LIN {X 0,Y 418.23,Z 297.388,A -85,B 0,C 180,E1 -10312.167,E2 -10312.167} C_VEL
LIN {X 0,Y 418.144,Z 297.404,A -85,B 0,C 180,E1 -10315.148,E2 -10315.148} C_VEL
LIN {X 0,Y 418.014,Z 297.572,A -85,B 0,C 180,E1 -10316.685,E2 -10316.685} C_VEL
LIN {X 0,Y 417.751,Z 304.24,A -85,B 0,C 180,E1 -10320.799,E2 -10320.799} C_VEL
LIN {X 0,Y 417.681,Z 309.464,A -85,B 0,C 180,E1 -10324.057,E2 -10324.057} C_VEL
LIN {X 0,Y 417.666,Z 315.525,A -85,B 0,C 180,E1 -10327.741,E2 -10327.741} C_VEL
LIN {X 0,Y 417.566,Z 321.841,A -85,B 0,C 180,E1 -10331.35,E2 -10331.35} C_VEL
LIN {X 0,Y 417.611,Z 324.668,A -85,B 0,C 180,E1 -10332.823,E2 -10332.823} C_VEL
LIN {X 0,Y 420.936,Z 337.978,A -85,B 0,C 180,E1 -10333.371,E2 -10333.371} C_VEL
LIN {X 0,Y 422.449,Z 346.002,A -85,B 0,C 180,E1 -10333.786,E2 -10333.786} C_VEL
LIN {X 0,Y 421.995,Z 357.531,A -85,B 0,C 180,E1 -10334.426,E2 -10334.426} C_VEL
LIN {X 0,Y 421.355,Z 369.434,A -85,B 0,C 180,E1 -10335.289,E2 -10335.289} C_VEL
LIN {X 0,Y 420.762,Z 379.905,A -85,B 0,C 180,E1 -10336.264,E2 -10336.264} C_VEL
LIN {X 0,Y 419.975,Z 390.066,A -85,B 0,C 180,E1 -10337.435,E2 -10337.435} C_VEL
LIN {X 0,Y 419.339,Z 398.59,A -85,B 0,C 180,E1 -10338.643,E2 -10338.643} C_VEL
LIN {X 0,Y 418.753,Z 406.88,A -85,B 0,C 180,E1 -10340.094,E2 -10340.094} C_VEL
LIN {X 0,Y 418.261,Z 412.53,A -85,B 0,C 180,E1 -10341.302,E2 -10341.302} C_VEL
LIN {X 0,Y 417.846,Z 418.534,A -85,B 0,C 180,E1 -10342.913,E2 -10342.913} C_VEL
LIN {X 0,Y 417.439,Z 423.536,A -85,B 0,C 180,E1 -10344.687,E2 -10344.687} C_VEL
LIN {X 0,Y 417.442,Z 426.435,A -85,B 0,C 180,E1 -10346.139,E2 -10346.139} C_VEL
LIN {X 0,Y 417.313,Z 427.849,A -85,B 0,C 180,E1 -10347.104,E2 -10347.104} C_VEL
LIN {X 0,Y 417.143,Z 429.456,A -85,B 0,C 180,E1 -10349.035,E2 -10349.035} C_VEL
LIN {X 0,Y 417.142,Z 429.69,A -85,B 0,C 180,E1 -10350,E2 -10350} C_VEL
LIN {X 0,Y 417.135,Z 429.529,A -85,B 0,C 180,E1 -10350.822,E2 -10350.822} C_VEL
LIN {X 0,Y 416.515,Z 429.25,A -85,B 0,C 180,E1 -10351.629,E2 -10351.629} C_VEL
LIN {X 0,Y 413.745,Z 428.239,A -85,B 0,C 180,E1 -10352.936,E2 -10352.936} C_VEL
LIN {X 0,Y 411.4,Z 426.873,A -85,B 0,C 180,E1 -10353.98,E2 -10353.98} C_VEL
LIN {X 0,Y 410.41,Z 425.491,A -85,B 0,C 180,E1 -10354.775,E2 -10354.775} C_VEL
LIN {X 0,Y 410.339,Z 424.938,A -85,B 0,C 180,E1 -10355.041,E2 -10355.041} C_VEL
LIN {X 0,Y 410.76,Z 420.293,A -85,B 0,C 180,E1 -10356.879,E2 -10356.879} C_VEL
LIN {X 0,Y 411.059,Z 415.281,A -85,B 0,C 180,E1 -10358.356,E2 -10358.356} C_VEL
LIN {X 0,Y 411.623,Z 408.945,A -85,B 0,C 180,E1 -10359.831,E2 -10359.831} C_VEL
LIN {X 0,Y 412.235,Z 401.072,A -85,B 0,C 180,E1 -10361.307,E2 -10361.307} C_VEL
LIN {X 0,Y 412.91,Z 393.024,A -85,B 0,C 180,E1 -10362.534,E2 -10362.534} C_VEL
LIN {X 0,Y 413.699,Z 383.148,A -85,B 0,C 180,E1 -10363.759,E2 -10363.759} C_VEL
LIN {X 0,Y 414.35,Z 372.025,A -85,B 0,C 180,E1 -10364.865,E2 -10364.865} C_VEL
LIN {X 0,Y 415.089,Z 361.127,A -85,B 0,C 180,E1 -10365.718,E2 -10365.718} C_VEL
LIN {X 0,Y 415.573,Z 349.447,A -85,B 0,C 180,E1 -10366.428,E2 -10366.428} C_VEL
LIN {X 0,Y 415.517,Z 345.816,A -85,B 0,C 180,E1 -10366.618,E2 -10366.618} C_VEL
LIN {X 0,Y 412.954,Z 334.164,A -85,B 0,C 180,E1 -10367.215,E2 -10367.215} C_VEL
LIN {X 0,Y 410.545,Z 324.943,A -85,B 0,C 180,E1 -10367.581,E2 -10367.581} C_VEL
LIN {X 0,Y 410.556,Z 320.487,A -85,B 0,C 180,E1 -10370.021,E2 -10370.021} C_VEL
LIN {X 0,Y 410.607,Z 315.08,A -85,B 0,C 180,E1 -10373.183,E2 -10373.183} C_VEL
LIN {X 0,Y 410.646,Z 309.763,A -85,B 0,C 180,E1 -10376.422,E2 -10376.422} C_VEL
LIN {X 0,Y 410.701,Z 304.45,A -85,B 0,C 180,E1 -10379.753,E2 -10379.753} C_VEL
LIN {X 0,Y 411.026,Z 298.292,A -85,B 0,C 180,E1 -10383.612,E2 -10383.612} C_VEL
LIN {X 0,Y 411.186,Z 298.268,A -85,B 0,C 180,E1 -10386.743,E2 -10386.743} C_VEL
LIN {X 0,Y 411.215,Z 298.265,A -85,B 0,C 180,E1 -10389.728,E2 -10389.728} C_VEL
LIN {X 0,Y 411.176,Z 298.27,A -85,B 0,C 180,E1 -10393.134,E2 -10393.134} C_VEL
LIN {X 0,Y 411.17,Z 298.27,A -85,B 0,C 180,E1 -10395.881,E2 -10395.881} C_VEL
LIN {X 0,Y 411.167,Z 298.268,A -85,B 0,C 180,E1 -10398.772,E2 -10398.772} C_VEL
LIN {X 0,Y 411.208,Z 298.262,A -85,B 0,C 180,E1 -10401.831,E2 -10401.831} C_VEL
LIN {X 0,Y 411.091,Z 298.276,A -85,B 0,C 180,E1 -10405.146,E2 -10405.146} C_VEL
LIN {X 0,Y 410.886,Z 298.336,A -85,B 0,C 180,E1 -10407.029,E2 -10407.029} C_VEL
LIN {X 0,Y 410.68,Z 304.557,A -85,B 0,C 180,E1 -10410.782,E2 -10410.782} C_VEL
LIN {X 0,Y 410.578,Z 309.184,A -85,B 0,C 180,E1 -10413.573,E2 -10413.573} C_VEL
LIN {X 0,Y 410.571,Z 312.781,A -85,B 0,C 180,E1 -10415.743,E2 -10415.743} C_VEL
LIN {X 0,Y 410.522,Z 318.015,A -85,B 0,C 180,E1 -10418.93,E2 -10418.93} C_VEL
LIN {X 0,Y 410.439,Z 323.255,A -85,B 0,C 180,E1 -10422.048,E2 -10422.048} C_VEL
LIN {X 0,Y 410.453,Z 325.126,A -85,B 0,C 180,E1 -10423.157,E2 -10423.157} C_VEL
LIN {X 0,Y 413.417,Z 339.31,A -85,B 0,C 180,E1 -10423.77,E2 -10423.77} C_VEL
LIN {X 0,Y 414.485,Z 345.44,A -85,B 0,C 180,E1 -10424.097,E2 -10424.097} C_VEL
LIN {X 0,Y 413.983,Z 356.751,A -85,B 0,C 180,E1 -10424.744,E2 -10424.744} C_VEL
LIN {X 0,Y 413.372,Z 368.988,A -85,B 0,C 180,E1 -10425.651,E2 -10425.651} C_VEL
LIN {X 0,Y 412.891,Z 380.326,A -85,B 0,C 180,E1 -10426.715,E2 -10426.715} C_VEL
LIN {X 0,Y 412.187,Z 390.845,A -85,B 0,C 180,E1 -10427.944,E2 -10427.944} C_VEL
LIN {X 0,Y 411.694,Z 399.473,A -85,B 0,C 180,E1 -10429.177,E2 -10429.177} C_VEL
LIN {X 0,Y 411.18,Z 407.897,A -85,B 0,C 180,E1 -10430.655,E2 -10430.655} C_VEL
LIN {X 0,Y 410.759,Z 414.655,A -85,B 0,C 180,E1 -10432.133,E2 -10432.133} C_VEL
LIN {X 0,Y 410.528,Z 420.608,A -85,B 0,C 180,E1 -10433.783,E2 -10433.783} C_VEL
LIN {X 0,Y 410.3,Z 424.235,A -85,B 0,C 180,E1 -10435.087,E2 -10435.087} C_VEL
LIN {X 0,Y 410.357,Z 426.377,A -85,B 0,C 180,E1 -10436.072,E2 -10436.072} C_VEL
LIN {X 0,Y 410.249,Z 428.088,A -85,B 0,C 180,E1 -10437.054,E2 -10437.054} C_VEL
LIN {X 0,Y 410.135,Z 429.383,A -85,B 0,C 180,E1 -10438.036,E2 -10438.036} C_VEL
LIN {X 0,Y 410.089,Z 430.201,A -85,B 0,C 180,E1 -10439.018,E2 -10439.018} C_VEL
LIN {X 0,Y 410.102,Z 430.614,A -85,B 0,C 180,E1 -10440,E2 -10440} C_VEL
LIN {X 0,Y 410.136,Z 430.622,A -85,B 0,C 180,E1 -10440.982,E2 -10440.982} C_VEL
LIN {X 0,Y 410.22,Z 430.164,A -85,B 0,C 180,E1 -10441.964,E2 -10441.964} C_VEL
LIN {X 0,Y 410.309,Z 429.298,A -85,B 0,C 180,E1 -10442.945,E2 -10442.945} C_VEL
LIN {X 0,Y 410.419,Z 428.027,A -85,B 0,C 180,E1 -10443.928,E2 -10443.928} C_VEL
LIN {X 0,Y 410.502,Z 425.256,A -85,B 0,C 180,E1 -10445.403,E2 -10445.403} C_VEL
LIN {X 0,Y 410.839,Z 421.383,A -85,B 0,C 180,E1 -10446.877,E2 -10446.877} C_VEL
LIN {X 0,Y 411.196,Z 416.313,A -85,B 0,C 180,E1 -10448.353,E2 -10448.353} C_VEL
LIN {X 0,Y 411.729,Z 409.882,A -85,B 0,C 180,E1 -10449.828,E2 -10449.828} C_VEL
LIN {X 0,Y 412.317,Z 401.876,A -85,B 0,C 180,E1 -10451.304,E2 -10451.304} C_VEL
LIN {X 0,Y 412.986,Z 391.822,A -85,B 0,C 180,E1 -10452.781,E2 -10452.781} C_VEL
LIN {X 0,Y 413.808,Z 382.015,A -85,B 0,C 180,E1 -10453.93,E2 -10453.93} C_VEL
LIN {X 0,Y 414.435,Z 371.233,A -85,B 0,C 180,E1 -10454.962,E2 -10454.962} C_VEL
LIN {X 0,Y 415.113,Z 359.685,A -85,B 0,C 180,E1 -10455.842,E2 -10455.842} C_VEL
LIN {X 0,Y 415.727,Z 346.23,A -85,B 0,C 180,E1 -10456.636,E2 -10456.636} C_VEL
LIN {X 0,Y 412.949,Z 334.877,A -85,B 0,C 180,E1 -10457.308,E2 -10457.308} C_VEL
LIN {X 0,Y 410.978,Z 328.466,A -85,B 0,C 180,E1 -10457.662,E2 -10457.662} C_VEL
LIN {X 0,Y 411.017,Z 322.663,A -85,B 0,C 180,E1 -10461.044,E2 -10461.044} C_VEL
LIN {X 0,Y 411.115,Z 317.021,A -85,B 0,C 180,E1 -10464.222,E2 -10464.222} C_VEL
LIN {X 0,Y 411.206,Z 309.985,A -85,B 0,C 180,E1 -10468.035,E2 -10468.035} C_VEL
LIN {X 0,Y 411.401,Z 303.588,A -85,B 0,C 180,E1 -10471.333,E2 -10471.333} C_VEL
LIN {X 0,Y 411.353,Z 299.92,A -85,B 0,C 180,E1 -10473.157,E2 -10473.157} C_VEL
LIN {X 0,Y 411.094,Z 298.282,A -85,B 0,C 180,E1 -10474.048,E2 -10474.048} C_VEL
LIN {X 0,Y 411.188,Z 298.268,A -85,B 0,C 180,E1 -10476.742,E2 -10476.742} C_VEL
LIN {X 0,Y 411.211,Z 298.264,A -85,B 0,C 180,E1 -10479.727,E2 -10479.727} C_VEL
LIN {X 0,Y 411.173,Z 298.271,A -85,B 0,C 180,E1 -10483.134,E2 -10483.134} C_VEL
LIN {X 0,Y 411.227,Z 298.412,A -85,B 0,C 180,E1 -10485.594,E2 -10485.594} C_VEL
LIN {X 0,Y 412.81,Z 306.462,A -85,B 0,C 180,E1 -10489.143,E2 -10489.143} C_VEL
LIN {X 0,Y 414.03,Z 312.933,A -85,B 0,C 180,E1 -10491.865,E2 -10491.865} C_VEL
LIN {X 0,Y 414.518,Z 317.262,A -85,B 0,C 180,E1 -10493.6,E2 -10493.6} C_VEL
LIN {X 0,Y 413.908,Z 324.461,A -85,B 0,C 180,E1 -10496.305,E2 -10496.305} C_VEL
LIN {X 0,Y 413.168,Z 334.07,A -85,B 0,C 180,E1 -10499.811,E2 -10499.811} C_VEL
LIN {X 0,Y 412.443,Z 343.508,A -85,B 0,C 180,E1 -10503.156,E2 -10503.156} C_VEL
LIN {X 0,Y 411.875,Z 352.746,A -85,B 0,C 180,E1 -10506.36,E2 -10506.36} C_VEL
LIN {X 0,Y 411.304,Z 363.53,A -85,B 0,C 180,E1 -10510.017,E2 -10510.017} C_VEL
LIN {X 0,Y 410.937,Z 370.534,A -85,B 0,C 180,E1 -10512.357,E2 -10512.357} C_VEL
LIN {X 0,Y 413.007,Z 384.417,A -85,B 0,C 180,E1 -10512.886,E2 -10512.886} C_VEL
LIN {X 0,Y 414.755,Z 397.429,A -85,B 0,C 180,E1 -10513.574,E2 -10513.574} C_VEL
LIN {X 0,Y 414.347,Z 408.316,A -85,B 0,C 180,E1 -10514.253,E2 -10514.253} C_VEL
LIN {X 0,Y 413.464,Z 420.652,A -85,B 0,C 180,E1 -10515.228,E2 -10515.228} C_VEL
LIN {X 0,Y 412.7,Z 431.639,A -85,B 0,C 180,E1 -10516.333,E2 -10516.333} C_VEL
LIN {X 0,Y 411.963,Z 442.383,A -85,B 0,C 180,E1 -10517.687,E2 -10517.687} C_VEL
LIN {X 0,Y 411.291,Z 450.345,A -85,B 0,C 180,E1 -10518.917,E2 -10518.917} C_VEL
LIN {X 0,Y 410.814,Z 458.183,A -85,B 0,C 180,E1 -10520.398,E2 -10520.398} C_VEL
LIN {X 0,Y 410.483,Z 463.52,A -85,B 0,C 180,E1 -10521.632,E2 -10521.632} C_VEL
LIN {X 0,Y 410.253,Z 468.725,A -85,B 0,C 180,E1 -10523.113,E2 -10523.113} C_VEL
LIN {X 0,Y 410.147,Z 472.759,A -85,B 0,C 180,E1 -10524.592,E2 -10524.592} C_VEL
LIN {X 0,Y 409.992,Z 475.719,A -85,B 0,C 180,E1 -10526.068,E2 -10526.068} C_VEL
LIN {X 0,Y 410.083,Z 477.145,A -85,B 0,C 180,E1 -10527.053,E2 -10527.053} C_VEL
LIN {X 0,Y 410.097,Z 478.729,A -85,B 0,C 180,E1 -10529.018,E2 -10529.018} C_VEL
LIN {X 0,Y 410.07,Z 478.915,A -85,B 0,C 180,E1 -10530,E2 -10530} C_VEL
LIN {X 0,Y 410.099,Z 478.658,A -85,B 0,C 180,E1 -10530.982,E2 -10530.982} C_VEL
LIN {X 0,Y 410.087,Z 476.91,A -85,B 0,C 180,E1 -10532.947,E2 -10532.947} C_VEL
LIN {X 0,Y 410.013,Z 475.412,A -85,B 0,C 180,E1 -10533.932,E2 -10533.932} C_VEL
LIN {X 0,Y 410.175,Z 472.315,A -85,B 0,C 180,E1 -10535.407,E2 -10535.407} C_VEL
LIN {X 0,Y 410.253,Z 468.131,A -85,B 0,C 180,E1 -10536.887,E2 -10536.887} C_VEL
LIN {X 0,Y 410.574,Z 461.734,A -85,B 0,C 180,E1 -10538.614,E2 -10538.614} C_VEL
LIN {X 0,Y 410.954,Z 454.778,A -85,B 0,C 180,E1 -10540.096,E2 -10540.096} C_VEL
LIN {X 0,Y 411.525,Z 446.209,A -85,B 0,C 180,E1 -10541.576,E2 -10541.576} C_VEL
LIN {X 0,Y 412.128,Z 437.452,A -85,B 0,C 180,E1 -10542.808,E2 -10542.808} C_VEL
LIN {X 0,Y 412.75,Z 427.734,A -85,B 0,C 180,E1 -10543.938,E2 -10543.938} C_VEL
LIN {X 0,Y 413.534,Z 416.299,A -85,B 0,C 180,E1 -10545.021,E2 -10545.021} C_VEL
LIN {X 0,Y 414.379,Z 405.059,A -85,B 0,C 180,E1 -10545.872,E2 -10545.872} C_VEL
LIN {X 0,Y 414.735,Z 398.212,A -85,B 0,C 180,E1 -10546.3,E2 -10546.3} C_VEL
LIN {X 0,Y 413.023,Z 384.848,A -85,B 0,C 180,E1 -10547.066,E2 -10547.066} C_VEL
LIN {X 0,Y 411.421,Z 371.369,A -85,B 0,C 180,E1 -10547.642,E2 -10547.642} C_VEL
LIN {X 0,Y 410.851,Z 367.765,A -85,B 0,C 180,E1 -10547.781,E2 -10547.781} C_VEL
LIN {X 0,Y 411.229,Z 357.761,A -85,B 0,C 180,E1 -10551.032,E2 -10551.032} C_VEL
LIN {X 0,Y 411.705,Z 348.288,A -85,B 0,C 180,E1 -10554.186,E2 -10554.186} C_VEL
LIN {X 0,Y 412.237,Z 338.537,A -85,B 0,C 180,E1 -10557.561,E2 -10557.561} C_VEL
LIN {X 0,Y 413.002,Z 328.602,A -85,B 0,C 180,E1 -10561.211,E2 -10561.211} C_VEL
LIN {X 0,Y 413.835,Z 319.926,A -85,B 0,C 180,E1 -10564.675,E2 -10564.675} C_VEL
LIN {X 0,Y 414.252,Z 315.928,A -85,B 0,C 180,E1 -10566.427,E2 -10566.427} C_VEL
LIN {X 0,Y 413.761,Z 311.596,A -85,B 0,C 180,E1 -10568.616,E2 -10568.616} C_VEL
LIN {X 0,Y 412.864,Z 306.663,A -85,B 0,C 180,E1 -10571.597,E2 -10571.597} C_VEL
LIN {X 0,Y 412.142,Z 303.106,A -85,B 0,C 180,E1 -10574.359,E2 -10574.359} C_VEL
LIN {X 0,Y 411.617,Z 300.463,A -85,B 0,C 180,E1 -10577.239,E2 -10577.239} C_VEL
LIN {X 0,Y 411.295,Z 298.828,A -85,B 0,C 180,E1 -10580.259,E2 -10580.259} C_VEL
LIN {X 0,Y 411.192,Z 298.267,A -85,B 0,C 180,E1 -10583.258,E2 -10583.258} C_VEL
LIN {X 0,Y 411.214,Z 298.311,A -85,B 0,C 180,E1 -10585.667,E2 -10585.667} C_VEL
LIN {X 0,Y 411.347,Z 299.206,A -85,B 0,C 180,E1 -10589.165,E2 -10589.165} C_VEL
LIN {X 0,Y 411.635,Z 300.67,A -85,B 0,C 180,E1 -10592.601,E2 -10592.601} C_VEL
LIN {X 0,Y 411.738,Z 302.464,A -85,B 0,C 180,E1 -10595.817,E2 -10595.817} C_VEL
LIN {X 0,Y 411.703,Z 303.825,A -85,B 0,C 180,E1 -10597.941,E2 -10597.941} C_VEL
LIN {X 0,Y 411.545,Z 306.033,A -85,B 0,C 180,E1 -10601.067,E2 -10601.067} C_VEL
LIN {X 0,Y 411.46,Z 307.135,A -85,B 0,C 180,E1 -10602.467,E2 -10602.467} C_VEL
LIN {X 0,Y 415.682,Z 319.179,A -85,B 0,C 180,E1 -10603.227,E2 -10603.227} C_VEL
LIN {X 0,Y 416.32,Z 321.604,A -85,B 0,C 180,E1 -10603.386,E2 -10603.386} C_VEL
LIN {X 0,Y 415.851,Z 333.205,A -85,B 0,C 180,E1 -10604.06,E2 -10604.06} C_VEL
LIN {X 0,Y 415.147,Z 345.588,A -85,B 0,C 180,E1 -10604.989,E2 -10604.989} C_VEL
LIN {X 0,Y 414.484,Z 356.455,A -85,B 0,C 180,E1 -10606.018,E2 -10606.018} C_VEL
LIN {X 0,Y 413.726,Z 366.834,A -85,B 0,C 180,E1 -10607.242,E2 -10607.242} C_VEL
LIN {X 0,Y 413.091,Z 375.295,A -85,B 0,C 180,E1 -10608.469,E2 -10608.469} C_VEL
LIN {X 0,Y 412.405,Z 383.502,A -85,B 0,C 180,E1 -10609.94,E2 -10609.94} C_VEL
LIN {X 0,Y 411.874,Z 390.158,A -85,B 0,C 180,E1 -10611.438,E2 -10611.438} C_VEL
LIN {X 0,Y 411.474,Z 394.915,A -85,B 0,C 180,E1 -10612.777,E2 -10612.777} C_VEL
LIN {X 0,Y 411.056,Z 398.678,A -85,B 0,C 180,E1 -10614.112,E2 -10614.112} C_VEL
LIN {X 0,Y 411.018,Z 400.837,A -85,B 0,C 180,E1 -10615.096,E2 -10615.096} C_VEL
LIN {X 0,Y 410.772,Z 402.572,A -85,B 0,C 180,E1 -10616.076,E2 -10616.076} C_VEL
LIN {X 0,Y 410.511,Z 403.832,A -85,B 0,C 180,E1 -10617.056,E2 -10617.056} C_VEL
LIN {X 0,Y 410.347,Z 404.677,A -85,B 0,C 180,E1 -10618.037,E2 -10618.037} C_VEL
LIN {X 0,Y 410.276,Z 405.113,A -85,B 0,C 180,E1 -10619.019,E2 -10619.019} C_VEL
LIN {X 0,Y 410.241,Z 405.1,A -85,B 0,C 180,E1 -10620,E2 -10620} C_VEL
LIN {X 0,Y 410.244,Z 404.668,A -85,B 0,C 180,E1 -10620.982,E2 -10620.982} C_VEL
LIN {X 0,Y 410.318,Z 403.834,A -85,B 0,C 180,E1 -10621.963,E2 -10621.963} C_VEL
LIN {X 0,Y 410.497,Z 402.572,A -85,B 0,C 180,E1 -10622.944,E2 -10622.944} C_VEL
LIN {X 0,Y 410.733,Z 399.85,A -85,B 0,C 180,E1 -10624.416,E2 -10624.416} C_VEL
LIN {X 0,Y 410.758,Z 396.102,A -85,B 0,C 180,E1 -10625.892,E2 -10625.892} C_VEL
LIN {X 0,Y 411.045,Z 391.08,A -85,B 0,C 180,E1 -10627.395,E2 -10627.395} C_VEL
LIN {X 0,Y 411.456,Z 383.804,A -85,B 0,C 180,E1 -10629.091,E2 -10629.091} C_VEL
LIN {X 0,Y 411.933,Z 375.802,A -85,B 0,C 180,E1 -10630.568,E2 -10630.568} C_VEL
LIN {X 0,Y 412.561,Z 365.797,A -85,B 0,C 180,E1 -10632.045,E2 -10632.045} C_VEL
LIN {X 0,Y 413.175,Z 355.451,A -85,B 0,C 180,E1 -10633.275,E2 -10633.275} C_VEL
LIN {X 0,Y 413.759,Z 343.258,A -85,B 0,C 180,E1 -10634.435,E2 -10634.435} C_VEL
LIN {X 0,Y 414.217,Z 332.568,A -85,B 0,C 180,E1 -10635.248,E2 -10635.248} C_VEL
LIN {X 0,Y 414.783,Z 319.92,A -85,B 0,C 180,E1 -10635.988,E2 -10635.988} C_VEL
LIN {X 0,Y 414.081,Z 315.24,A -85,B 0,C 180,E1 -10636.243,E2 -10636.243} C_VEL
LIN {X 0,Y 410.732,Z 301.39,A -85,B 0,C 180,E1 -10636.892,E2 -10636.892} C_VEL
LIN {X 0,Y 410.516,Z 300.22,A -85,B 0,C 180,E1 -10636.952,E2 -10636.952} C_VEL
LIN {X 0,Y 410.442,Z 299.006,A -85,B 0,C 180,E1 -10637.952,E2 -10637.952} C_VEL
LIN {X 0,Y 410.56,Z 298.347,A -85,B 0,C 180,E1 -10638.98,E2 -10638.98} C_VEL
LIN {X 0,Y 410.936,Z 298.298,A -85,B 0,C 180,E1 -10642.551,E2 -10642.551} C_VEL
LIN {X 0,Y 411.164,Z 298.264,A -85,B 0,C 180,E1 -10645.298,E2 -10645.298} C_VEL
LIN {X 0,Y 411.243,Z 298.254,A -85,B 0,C 180,E1 -10647.479,E2 -10647.479} C_VEL
LIN {X 0,Y 411.192,Z 298.26,A -85,B 0,C 180,E1 -10650.848,E2 -10650.848} C_VEL
LIN {X 0,Y 411.209,Z 298.263,A -85,B 0,C 180,E1 -10654.333,E2 -10654.333} C_VEL
LIN {X 0,Y 411.197,Z 298.269,A -85,B 0,C 180,E1 -10657.974,E2 -10657.974} C_VEL
LIN {X 0,Y 411.166,Z 298.269,A -85,B 0,C 180,E1 -10661.228,E2 -10661.228} C_VEL
LIN {X 0,Y 411.18,Z 298.265,A -85,B 0,C 180,E1 -10664.49,E2 -10664.49} C_VEL
LIN {X 0,Y 411.18,Z 298.266,A -85,B 0,C 180,E1 -10668.195,E2 -10668.195} C_VEL
LIN {X 0,Y 411.22,Z 298.261,A -85,B 0,C 180,E1 -10670.776,E2 -10670.776} C_VEL
LIN {X 0,Y 411.187,Z 298.269,A -85,B 0,C 180,E1 -10673.449,E2 -10673.449} C_VEL
LIN {X 0,Y 410.989,Z 298.381,A -85,B 0,C 180,E1 -10676.604,E2 -10676.604} C_VEL
LIN {X 0,Y 410.732,Z 305.091,A -85,B 0,C 180,E1 -10680.769,E2 -10680.769} C_VEL
LIN {X 0,Y 410.646,Z 309.599,A -85,B 0,C 180,E1 -10683.578,E2 -10683.578} C_VEL
LIN {X 0,Y 410.607,Z 314.889,A -85,B 0,C 180,E1 -10686.817,E2 -10686.817} C_VEL
LIN {X 0,Y 410.595,Z 320.851,A -85,B 0,C 180,E1 -10690.291,E2 -10690.291} C_VEL
LIN {X 0,Y 410.564,Z 324.92,A -85,B 0,C 180,E1 -10692.504,E2 -10692.504} C_VEL
LIN {X 0,Y 414.246,Z 339.604,A -85,B 0,C 180,E1 -10693.142,E2 -10693.142} C_VEL
LIN {X 0,Y 415.607,Z 347.386,A -85,B 0,C 180,E1 -10693.563,E2 -10693.563} C_VEL
LIN {X 0,Y 415.087,Z 359.759,A -85,B 0,C 180,E1 -10694.282,E2 -10694.282} C_VEL
LIN {X 0,Y 414.393,Z 371.394,A -85,B 0,C 180,E1 -10695.175,E2 -10695.175} C_VEL
LIN {X 0,Y 413.71,Z 382.276,A -85,B 0,C 180,E1 -10696.242,E2 -10696.242} C_VEL
LIN {X 0,Y 412.944,Z 392.35,A -85,B 0,C 180,E1 -10697.467,E2 -10697.467} C_VEL
LIN {X 0,Y 412.185,Z 401.962,A -85,B 0,C 180,E1 -10698.941,E2 -10698.941} C_VEL
LIN {X 0,Y 411.537,Z 409.688,A -85,B 0,C 180,E1 -10700.415,E2 -10700.415} C_VEL
LIN {X 0,Y 411.119,Z 414.904,A -85,B 0,C 180,E1 -10701.645,E2 -10701.645} C_VEL
LIN {X 0,Y 410.76,Z 420,A -85,B 0,C 180,E1 -10703.121,E2 -10703.121} C_VEL
LIN {X 0,Y 410.383,Z 423.951,A -85,B 0,C 180,E1 -10704.595,E2 -10704.595} C_VEL
LIN {X 0,Y 410.386,Z 426.85,A -85,B 0,C 180,E1 -10706.072,E2 -10706.072} C_VEL
LIN {X 0,Y 410.25,Z 428.264,A -85,B 0,C 180,E1 -10707.054,E2 -10707.054} C_VEL
LIN {X 0,Y 410.062,Z 429.871,A -85,B 0,C 180,E1 -10709.018,E2 -10709.018} C_VEL
LIN {X 0,Y 410.057,Z 430.104,A -85,B 0,C 180,E1 -10710,E2 -10710} C_VEL
LIN {X 0,Y 410.135,Z 429.332,A -85,B 0,C 180,E1 -10711.964,E2 -10711.964} C_VEL
LIN {X 0,Y 410.249,Z 428.368,A -85,B 0,C 180,E1 -10712.946,E2 -10712.946} C_VEL
LIN {X 0,Y 410.378,Z 427.012,A -85,B 0,C 180,E1 -10713.928,E2 -10713.928} C_VEL
LIN {X 0,Y 410.339,Z 424.938,A -85,B 0,C 180,E1 -10715.041,E2 -10715.041} C_VEL
LIN {X 0,Y 409.757,Z 423.224,A -85,B 0,C 180,E1 -10715.828,E2 -10715.828} C_VEL
LIN {X 0,Y 407.185,Z 420.047,A -85,B 0,C 180,E1 -10717.097,E2 -10717.097} C_VEL
LIN {X 0,Y 404.697,Z 416.203,A -85,B 0,C 180,E1 -10718.34,E2 -10718.34} C_VEL
LIN {X 0,Y 404.251,Z 413.42,A -85,B 0,C 180,E1 -10719.078,E2 -10719.078} C_VEL
LIN {X 0,Y 404.867,Z 406.94,A -85,B 0,C 180,E1 -10720.502,E2 -10720.502} C_VEL
LIN {X 0,Y 405.569,Z 398.435,A -85,B 0,C 180,E1 -10722.002,E2 -10722.002} C_VEL
LIN {X 0,Y 406.367,Z 389.716,A -85,B 0,C 180,E1 -10723.247,E2 -10723.247} C_VEL
LIN {X 0,Y 407.019,Z 380.308,A -85,B 0,C 180,E1 -10724.354,E2 -10724.354} C_VEL
LIN {X 0,Y 407.695,Z 369.564,A -85,B 0,C 180,E1 -10725.369,E2 -10725.369} C_VEL
LIN {X 0,Y 408.447,Z 358.139,A -85,B 0,C 180,E1 -10726.213,E2 -10726.213} C_VEL
LIN {X 0,Y 408.727,Z 347.121,A -85,B 0,C 180,E1 -10726.853,E2 -10726.853} C_VEL
LIN {X 0,Y 405.966,Z 334.5,A -85,B 0,C 180,E1 -10727.521,E2 -10727.521} C_VEL
LIN {X 0,Y 403.51,Z 325.248,A -85,B 0,C 180,E1 -10727.928,E2 -10727.928} C_VEL
LIN {X 0,Y 403.501,Z 320.783,A -85,B 0,C 180,E1 -10730.387,E2 -10730.387} C_VEL
LIN {X 0,Y 403.562,Z 315.298,A -85,B 0,C 180,E1 -10733.612,E2 -10733.612} C_VEL
LIN {X 0,Y 403.638,Z 309.177,A -85,B 0,C 180,E1 -10737.377,E2 -10737.377} C_VEL
LIN {X 0,Y 403.7,Z 304.485,A -85,B 0,C 180,E1 -10740.322,E2 -10740.322} C_VEL
LIN {X 0,Y 403.995,Z 299.167,A -85,B 0,C 180,E1 -10743.688,E2 -10743.688} C_VEL
LIN {X 0,Y 404.133,Z 299.147,A -85,B 0,C 180,E1 -10746.874,E2 -10746.874} C_VEL
LIN {X 0,Y 404.15,Z 299.145,A -85,B 0,C 180,E1 -10750.08,E2 -10750.08} C_VEL
LIN {X 0,Y 404.155,Z 299.145,A -85,B 0,C 180,E1 -10753.084,E2 -10753.084} C_VEL
LIN {X 0,Y 404.15,Z 299.144,A -85,B 0,C 180,E1 -10755.926,E2 -10755.926} C_VEL
LIN {X 0,Y 404.122,Z 299.146,A -85,B 0,C 180,E1 -10758.635,E2 -10758.635} C_VEL
LIN {X 0,Y 404.157,Z 299.14,A -85,B 0,C 180,E1 -10761.492,E2 -10761.492} C_VEL
LIN {X 0,Y 404.058,Z 299.152,A -85,B 0,C 180,E1 -10764.971,E2 -10764.971} C_VEL
LIN {X 0,Y 403.845,Z 299.325,A -85,B 0,C 180,E1 -10767.109,E2 -10767.109} C_VEL
LIN {X 0,Y 403.628,Z 305.437,A -85,B 0,C 180,E1 -10770.821,E2 -10770.821} C_VEL
LIN {X 0,Y 403.514,Z 310.989,A -85,B 0,C 180,E1 -10774.187,E2 -10774.187} C_VEL
LIN {X 0,Y 403.484,Z 316.391,A -85,B 0,C 180,E1 -10777.468,E2 -10777.468} C_VEL
LIN {X 0,Y 403.459,Z 321.702,A -85,B 0,C 180,E1 -10780.672,E2 -10780.672} C_VEL
LIN {X 0,Y 403.396,Z 325.469,A -85,B 0,C 180,E1 -10782.931,E2 -10782.931} C_VEL
LIN {X 0,Y 405.999,Z 337.78,A -85,B 0,C 180,E1 -10783.455,E2 -10783.455} C_VEL
LIN {X 0,Y 407.556,Z 346.315,A -85,B 0,C 180,E1 -10783.918,E2 -10783.918} C_VEL
LIN {X 0,Y 407.015,Z 357.948,A -85,B 0,C 180,E1 -10784.604,E2 -10784.604} C_VEL
LIN {X 0,Y 406.312,Z 370.998,A -85,B 0,C 180,E1 -10785.613,E2 -10785.613} C_VEL
LIN {X 0,Y 405.788,Z 382.335,A -85,B 0,C 180,E1 -10786.733,E2 -10786.733} C_VEL
LIN {X 0,Y 405.08,Z 392.598,A -85,B 0,C 180,E1 -10787.983,E2 -10787.983} C_VEL
LIN {X 0,Y 404.595,Z 401.012,A -85,B 0,C 180,E1 -10789.238,E2 -10789.238} C_VEL
LIN {X 0,Y 404.076,Z 409.206,A -85,B 0,C 180,E1 -10790.742,E2 -10790.742} C_VEL
LIN {X 0,Y 403.735,Z 414.81,A -85,B 0,C 180,E1 -10791.995,E2 -10791.995} C_VEL
LIN {X 0,Y 403.494,Z 420.111,A -85,B 0,C 180,E1 -10793.45,E2 -10793.45} C_VEL
LIN {X 0,Y 403.231,Z 424.518,A -85,B 0,C 180,E1 -10795,E2 -10795} C_VEL
LIN {X 0,Y 403.272,Z 426.71,A -85,B 0,C 180,E1 -10796.003,E2 -10796.003} C_VEL
LIN {X 0,Y 403.188,Z 428.443,A -85,B 0,C 180,E1 -10797.002,E2 -10797.002} C_VEL
LIN {X 0,Y 403.064,Z 429.768,A -85,B 0,C 180,E1 -10798.001,E2 -10798.001} C_VEL
LIN {X 0,Y 403.009,Z 430.626,A -85,B 0,C 180,E1 -10799.001,E2 -10799.001} C_VEL
LIN {X 0,Y 403.018,Z 431.061,A -85,B 0,C 180,E1 -10800,E2 -10800} C_VEL
LIN {X 0,Y 403.053,Z 431.099,A -85,B 0,C 180,E1 -10800.999,E2 -10800.999} C_VEL
LIN {X 0,Y 403.143,Z 430.678,A -85,B 0,C 180,E1 -10801.998,E2 -10801.998} C_VEL
LIN {X 0,Y 403.245,Z 429.832,A -85,B 0,C 180,E1 -10802.997,E2 -10802.997} C_VEL
LIN {X 0,Y 403.373,Z 428.581,A -85,B 0,C 180,E1 -10803.996,E2 -10803.996} C_VEL
LIN {X 0,Y 403.456,Z 425.848,A -85,B 0,C 180,E1 -10805.498,E2 -10805.498} C_VEL
LIN {X 0,Y 403.892,Z 421.002,A -85,B 0,C 180,E1 -10807.323,E2 -10807.323} C_VEL
LIN {X 0,Y 404.409,Z 415.048,A -85,B 0,C 180,E1 -10808.998,E2 -10808.998} C_VEL
LIN {X 0,Y 404.977,Z 408.173,A -85,B 0,C 180,E1 -10810.499,E2 -10810.499} C_VEL
LIN {X 0,Y 405.638,Z 399.612,A -85,B 0,C 180,E1 -10812,E2 -10812} C_VEL
LIN {X 0,Y 406.383,Z 390.763,A -85,B 0,C 180,E1 -10813.247,E2 -10813.247} C_VEL
LIN {X 0,Y 407.212,Z 379.809,A -85,B 0,C 180,E1 -10814.507,E2 -10814.507} C_VEL
LIN {X 0,Y 407.88,Z 369.209,A -85,B 0,C 180,E1 -10815.49,E2 -10815.49} C_VEL
LIN {X 0,Y 408.594,Z 357.572,A -85,B 0,C 180,E1 -10816.348,E2 -10816.348} C_VEL
LIN {X 0,Y 409.123,Z 348.106,A -85,B 0,C 180,E1 -10816.902,E2 -10816.902} C_VEL
LIN {X 0,Y 406.438,Z 336.838,A -85,B 0,C 180,E1 -10817.611,E2 -10817.611} C_VEL
LIN {X 0,Y 403.997,Z 329.018,A -85,B 0,C 180,E1 -10818.084,E2 -10818.084} C_VEL
LIN {X 0,Y 404.04,Z 325.149,A -85,B 0,C 180,E1 -10820.358,E2 -10820.358} C_VEL
LIN {X 0,Y 404.125,Z 319.566,A -85,B 0,C 180,E1 -10823.577,E2 -10823.577} C_VEL
LIN {X 0,Y 404.197,Z 313.631,A -85,B 0,C 180,E1 -10826.877,E2 -10826.877} C_VEL
LIN {X 0,Y 404.426,Z 307.299,A -85,B 0,C 180,E1 -10830.262,E2 -10830.262} C_VEL
LIN {X 0,Y 404.524,Z 302.761,A -85,B 0,C 180,E1 -10832.587,E2 -10832.587} C_VEL
LIN {X 0,Y 404.066,Z 299.158,A -85,B 0,C 180,E1 -10834.573,E2 -10834.573} C_VEL
LIN {X 0,Y 404.142,Z 299.145,A -85,B 0,C 180,E1 -10837.492,E2 -10837.492} C_VEL
LIN {X 0,Y 404.149,Z 299.145,A -85,B 0,C 180,E1 -10840.08,E2 -10840.08} C_VEL
LIN {X 0,Y 404.152,Z 299.145,A -85,B 0,C 180,E1 -10843.083,E2 -10843.083} C_VEL
LIN {X 0,Y 404.169,Z 299.242,A -85,B 0,C 180,E1 -10845.213,E2 -10845.213} C_VEL
LIN {X 0,Y 405.442,Z 305.847,A -85,B 0,C 180,E1 -10848.191,E2 -10848.191} C_VEL
LIN {X 0,Y 406.979,Z 313.657,A -85,B 0,C 180,E1 -10851.561,E2 -10851.561} C_VEL
LIN {X 0,Y 407.556,Z 318.378,A -85,B 0,C 180,E1 -10853.492,E2 -10853.492} C_VEL
LIN {X 0,Y 406.848,Z 326.113,A -85,B 0,C 180,E1 -10856.442,E2 -10856.442} C_VEL
LIN {X 0,Y 406.11,Z 335.475,A -85,B 0,C 180,E1 -10859.915,E2 -10859.915} C_VEL
LIN {X 0,Y 405.265,Z 346.155,A -85,B 0,C 180,E1 -10863.755,E2 -10863.755} C_VEL
LIN {X 0,Y 404.805,Z 353.857,A -85,B 0,C 180,E1 -10866.465,E2 -10866.465} C_VEL
LIN {X 0,Y 404.165,Z 364.865,A -85,B 0,C 180,E1 -10870.275,E2 -10870.275} C_VEL
LIN {X 0,Y 403.901,Z 370.036,A -85,B 0,C 180,E1 -10872.043,E2 -10872.043} C_VEL
LIN {X 0,Y 406.085,Z 384.87,A -85,B 0,C 180,E1 -10872.63,E2 -10872.63} C_VEL
LIN {X 0,Y 407.787,Z 397.869,A -85,B 0,C 180,E1 -10873.35,E2 -10873.35} C_VEL
LIN {X 0,Y 407.74,Z 404.003,A -85,B 0,C 180,E1 -10873.734,E2 -10873.734} C_VEL
LIN {X 0,Y 406.885,Z 415.744,A -85,B 0,C 180,E1 -10874.599,E2 -10874.599} C_VEL
LIN {X 0,Y 406.074,Z 426.413,A -85,B 0,C 180,E1 -10875.594,E2 -10875.594} C_VEL
LIN {X 0,Y 405.387,Z 436.187,A -85,B 0,C 180,E1 -10876.722,E2 -10876.722} C_VEL
LIN {X 0,Y 404.672,Z 445.102,A -85,B 0,C 180,E1 -10877.971,E2 -10877.971} C_VEL
LIN {X 0,Y 403.999,Z 453.863,A -85,B 0,C 180,E1 -10879.475,E2 -10879.475} C_VEL
LIN {X 0,Y 403.56,Z 460.884,A -85,B 0,C 180,E1 -10880.983,E2 -10880.983} C_VEL
LIN {X 0,Y 403.211,Z 466.502,A -85,B 0,C 180,E1 -10882.488,E2 -10882.488} C_VEL
LIN {X 0,Y 403.069,Z 470.919,A -85,B 0,C 180,E1 -10883.995,E2 -10883.995} C_VEL
LIN {X 0,Y 403.044,Z 473.249,A -85,B 0,C 180,E1 -10884.998,E2 -10884.998} C_VEL
LIN {X 0,Y 402.912,Z 475.129,A -85,B 0,C 180,E1 -10885.999,E2 -10885.999} C_VEL
LIN {X 0,Y 403.018,Z 476.558,A -85,B 0,C 180,E1 -10887.001,E2 -10887.001} C_VEL
LIN {X 0,Y 403.044,Z 478.14,A -85,B 0,C 180,E1 -10889.001,E2 -10889.001} C_VEL
LIN {X 0,Y 403.018,Z 478.323,A -85,B 0,C 180,E1 -10890,E2 -10890} C_VEL
LIN {X 0,Y 403.047,Z 478.062,A -85,B 0,C 180,E1 -10890.999,E2 -10890.999} C_VEL
LIN {X 0,Y 403.024,Z 476.3,A -85,B 0,C 180,E1 -10892.999,E2 -10892.999} C_VEL
LIN {X 0,Y 402.933,Z 474.79,A -85,B 0,C 180,E1 -10894.001,E2 -10894.001} C_VEL
LIN {X 0,Y 403.093,Z 471.678,A -85,B 0,C 180,E1 -10895.503,E2 -10895.503} C_VEL
LIN {X 0,Y 403.186,Z 467.48,A -85,B 0,C 180,E1 -10897.009,E2 -10897.009} C_VEL
LIN {X 0,Y 403.527,Z 461.077,A -85,B 0,C 180,E1 -10898.766,E2 -10898.766} C_VEL
LIN {X 0,Y 403.896,Z 454.142,A -85,B 0,C 180,E1 -10900.274,E2 -10900.274} C_VEL
LIN {X 0,Y 404.508,Z 445.548,A -85,B 0,C 180,E1 -10901.78,E2 -10901.78} C_VEL
LIN {X 0,Y 405.181,Z 436.824,A -85,B 0,C 180,E1 -10903.032,E2 -10903.032} C_VEL
LIN {X 0,Y 405.868,Z 426.416,A -85,B 0,C 180,E1 -10904.26,E2 -10904.26} C_VEL
LIN {X 0,Y 406.755,Z 414.379,A -85,B 0,C 180,E1 -10905.406,E2 -10905.406} C_VEL
LIN {X 0,Y 407.631,Z 402.823,A -85,B 0,C 180,E1 -10906.27,E2 -10906.27} C_VEL
LIN {X 0,Y 407.735,Z 397.959,A -85,B 0,C 180,E1 -10906.588,E2 -10906.588} C_VEL
LIN {X 0,Y 406.238,Z 385.682,A -85,B 0,C 180,E1 -10907.328,E2 -10907.328} C_VEL
LIN {X 0,Y 404.678,Z 372.195,A -85,B 0,C 180,E1 -10907.951,E2 -10907.951} C_VEL
LIN {X 0,Y 403.813,Z 366.974,A -85,B 0,C 180,E1 -10908.162,E2 -10908.162} C_VEL
LIN {X 0,Y 404.22,Z 357.201,A -85,B 0,C 180,E1 -10911.415,E2 -10911.415} C_VEL
LIN {X 0,Y 404.724,Z 347.808,A -85,B 0,C 180,E1 -10914.63,E2 -10914.63} C_VEL
LIN {X 0,Y 405.268,Z 338.595,A -85,B 0,C 180,E1 -10917.919,E2 -10917.919} C_VEL
LIN {X 0,Y 406.025,Z 329.682,A -85,B 0,C 180,E1 -10921.284,E2 -10921.284} C_VEL
LIN {X 0,Y 407.053,Z 320.071,A -85,B 0,C 180,E1 -10925.265,E2 -10925.265} C_VEL
LIN {X 0,Y 407.292,Z 316.024,A -85,B 0,C 180,E1 -10927.153,E2 -10927.153} C_VEL
LIN {X 0,Y 406.504,Z 311.311,A -85,B 0,C 180,E1 -10929.769,E2 -10929.769} C_VEL
LIN {X 0,Y 405.725,Z 307.251,A -85,B 0,C 180,E1 -10932.498,E2 -10932.498} C_VEL
LIN {X 0,Y 405.105,Z 303.982,A -85,B 0,C 180,E1 -10935.34,E2 -10935.34} C_VEL
LIN {X 0,Y 404.636,Z 301.661,A -85,B 0,C 180,E1 -10938.319,E2 -10938.319} C_VEL
LIN {X 0,Y 404.393,Z 300.316,A -85,B 0,C 180,E1 -10941.45,E2 -10941.45} C_VEL
LIN {X 0,Y 404.324,Z 299.963,A -85,B 0,C 180,E1 -10944.782,E2 -10944.782} C_VEL
LIN {X 0,Y 404.412,Z 300.571,A -85,B 0,C 180,E1 -10948.38,E2 -10948.38} C_VEL
LIN {X 0,Y 404.565,Z 301.43,A -85,B 0,C 180,E1 -10950.895,E2 -10950.895} C_VEL
LIN {X 0,Y 404.734,Z 302.44,A -85,B 0,C 180,E1 -10953.161,E2 -10953.161} C_VEL
LIN {X 0,Y 404.763,Z 303.633,A -85,B 0,C 180,E1 -10955.372,E2 -10955.372} C_VEL
LIN {X 0,Y 404.742,Z 304.939,A -85,B 0,C 180,E1 -10957.542,E2 -10957.542} C_VEL
LIN {X 0,Y 404.587,Z 307.096,A -85,B 0,C 180,E1 -10960.728,E2 -10960.728} C_VEL
LIN {X 0,Y 404.53,Z 308.26,A -85,B 0,C 180,E1 -10962.064,E2 -10962.064} C_VEL
LIN {X 0,Y 409.001,Z 320.719,A -85,B 0,C 180,E1 -10962.909,E2 -10962.909} C_VEL
LIN {X 0,Y 409.718,Z 323.707,A -85,B 0,C 180,E1 -10963.11,E2 -10963.11} C_VEL
LIN {X 0,Y 409.085,Z 336.772,A -85,B 0,C 180,E1 -10963.917,E2 -10963.917} C_VEL
LIN {X 0,Y 408.329,Z 348.819,A -85,B 0,C 180,E1 -10964.885,E2 -10964.885} C_VEL
LIN {X 0,Y 407.511,Z 360.029,A -85,B 0,C 180,E1 -10966.028,E2 -10966.028} C_VEL
LIN {X 0,Y 406.746,Z 369.839,A -85,B 0,C 180,E1 -10967.273,E2 -10967.273} C_VEL
LIN {X 0,Y 406.089,Z 377.887,A -85,B 0,C 180,E1 -10968.52,E2 -10968.52} C_VEL
LIN {X 0,Y 405.323,Z 385.761,A -85,B 0,C 180,E1 -10970.015,E2 -10970.015} C_VEL
LIN {X 0,Y 404.861,Z 392.202,A -85,B 0,C 180,E1 -10971.565,E2 -10971.565} C_VEL
LIN {X 0,Y 404.255,Z 396.955,A -85,B 0,C 180,E1 -10973.01,E2 -10973.01} C_VEL
LIN {X 0,Y 404.035,Z 400.688,A -85,B 0,C 180,E1 -10974.51,E2 -10974.51} C_VEL
LIN {X 0,Y 403.746,Z 403.388,A -85,B 0,C 180,E1 -10976.007,E2 -10976.007} C_VEL
LIN {X 0,Y 403.473,Z 404.625,A -85,B 0,C 180,E1 -10977.005,E2 -10977.005} C_VEL
LIN {X 0,Y 403.296,Z 405.446,A -85,B 0,C 180,E1 -10978.003,E2 -10978.003} C_VEL
LIN {X 0,Y 403.217,Z 405.852,A -85,B 0,C 180,E1 -10979.001,E2 -10979.001} C_VEL
LIN {X 0,Y 403.18,Z 405.8,A -85,B 0,C 180,E1 -10980,E2 -10980} C_VEL
LIN {X 0,Y 403.186,Z 405.341,A -85,B 0,C 180,E1 -10980.999,E2 -10980.999} C_VEL
LIN {X 0,Y 403.269,Z 404.473,A -85,B 0,C 180,E1 -10981.998,E2 -10981.998} C_VEL
LIN {X 0,Y 403.457,Z 403.161,A -85,B 0,C 180,E1 -10982.996,E2 -10982.996} C_VEL
LIN {X 0,Y 403.673,Z 400.385,A -85,B 0,C 180,E1 -10984.494,E2 -10984.494} C_VEL
LIN {X 0,Y 403.701,Z 396.575,A -85,B 0,C 180,E1 -10985.996,E2 -10985.996} C_VEL
LIN {X 0,Y 404.047,Z 390.747,A -85,B 0,C 180,E1 -10987.718,E2 -10987.718} C_VEL
LIN {X 0,Y 404.455,Z 384.134,A -85,B 0,C 180,E1 -10989.249,E2 -10989.249} C_VEL
LIN {X 0,Y 404.941,Z 376.014,A -85,B 0,C 180,E1 -10990.753,E2 -10990.753} C_VEL
LIN {X 0,Y 405.592,Z 365.906,A -85,B 0,C 180,E1 -10992.255,E2 -10992.255} C_VEL
LIN {X 0,Y 406.244,Z 355.393,A -85,B 0,C 180,E1 -10993.506,E2 -10993.506} C_VEL
LIN {X 0,Y 406.789,Z 344.265,A -85,B 0,C 180,E1 -10994.58,E2 -10994.58} C_VEL
LIN {X 0,Y 407.326,Z 332.108,A -85,B 0,C 180,E1 -10995.512,E2 -10995.512} C_VEL
LIN {X 0,Y 407.847,Z 319.978,A -85,B 0,C 180,E1 -10996.225,E2 -10996.225} C_VEL
LIN {X 0,Y 404.876,Z 306.729,A -85,B 0,C 180,E1 -10996.923,E2 -10996.923} C_VEL
LIN {X 0,Y 403.486,Z 300.794,A -85,B 0,C 180,E1 -10997.181,E2 -10997.181} C_VEL
LIN {X 0,Y 403.408,Z 299.441,A -85,B 0,C 180,E1 -10998.276,E2 -10998.276} C_VEL
LIN {X 0,Y 403.658,Z 299.204,A -85,B 0,C 180,E1 -11000.378,E2 -11000.378} C_VEL
LIN {X 0,Y 403.98,Z 299.166,A -85,B 0,C 180,E1 -11003.586,E2 -11003.586} C_VEL
LIN {X 0,Y 404.137,Z 299.138,A -85,B 0,C 180,E1 -11005.77,E2 -11005.77} C_VEL
LIN {X 0,Y 404.189,Z 299.134,A -85,B 0,C 180,E1 -11008,E2 -11008} C_VEL
LIN {X 0,Y 404.142,Z 299.136,A -85,B 0,C 180,E1 -11011.558,E2 -11011.558} C_VEL
LIN {X 0,Y 404.187,Z 299.131,A -85,B 0,C 180,E1 -11015.016,E2 -11015.016} C_VEL
LIN {X 0,Y 404.157,Z 299.14,A -85,B 0,C 180,E1 -11018.757,E2 -11018.757} C_VEL
LIN {X 0,Y 404.126,Z 299.148,A -85,B 0,C 180,E1 -11021.6,E2 -11021.6} C_VEL
LIN {X 0,Y 404.15,Z 299.141,A -85,B 0,C 180,E1 -11024.522,E2 -11024.522} C_VEL
LIN {X 0,Y 404.139,Z 299.142,A -85,B 0,C 180,E1 -11027.296,E2 -11027.296} C_VEL
LIN {X 0,Y 404.171,Z 299.141,A -85,B 0,C 180,E1 -11029.955,E2 -11029.955} C_VEL
LIN {X 0,Y 404.133,Z 299.145,A -85,B 0,C 180,E1 -11033.126,E2 -11033.126} C_VEL
LIN {X 0,Y 403.973,Z 299.168,A -85,B 0,C 180,E1 -11036.479,E2 -11036.479} C_VEL
LIN {X 0,Y 403.709,Z 306.136,A -85,B 0,C 180,E1 -11040.827,E2 -11040.827} C_VEL
LIN {X 0,Y 403.59,Z 311.524,A -85,B 0,C 180,E1 -11044.193,E2 -11044.193} C_VEL
LIN {X 0,Y 403.583,Z 316.918,A -85,B 0,C 180,E1 -11047.474,E2 -11047.474} C_VEL
LIN {X 0,Y 403.523,Z 322.481,A -85,B 0,C 180,E1 -11050.676,E2 -11050.676} C_VEL
LIN {X 0,Y 403.531,Z 325.326,A -85,B 0,C 180,E1 -11052.202,E2 -11052.202} C_VEL
LIN {X 0,Y 406.917,Z 338.548,A -85,B 0,C 180,E1 -11052.772,E2 -11052.772} C_VEL
LIN {X 0,Y 408.819,Z 348.118,A -85,B 0,C 180,E1 -11053.3,E2 -11053.3} C_VEL
LIN {X 0,Y 408.288,Z 360.156,A -85,B 0,C 180,E1 -11054.013,E2 -11054.013} C_VEL
LIN {X 0,Y 407.69,Z 370.241,A -85,B 0,C 180,E1 -11054.784,E2 -11054.784} C_VEL
LIN {X 0,Y 407.007,Z 380.938,A -85,B 0,C 180,E1 -11055.814,E2 -11055.814} C_VEL
LIN {X 0,Y 406.192,Z 390.885,A -85,B 0,C 180,E1 -11057.001,E2 -11057.001} C_VEL
LIN {X 0,Y 405.477,Z 399.413,A -85,B 0,C 180,E1 -11058.249,E2 -11058.249} C_VEL
LIN {X 0,Y 404.783,Z 407.708,A -85,B 0,C 180,E1 -11059.749,E2 -11059.749} C_VEL
LIN {X 0,Y 404.265,Z 413.358,A -85,B 0,C 180,E1 -11060.998,E2 -11060.998} C_VEL
LIN {X 0,Y 403.749,Z 419.904,A -85,B 0,C 180,E1 -11062.837,E2 -11062.837} C_VEL
LIN {X 0,Y 403.334,Z 424.366,A -85,B 0,C 180,E1 -11064.501,E2 -11064.501} C_VEL
LIN {X 0,Y 403.311,Z 427.265,A -85,B 0,C 180,E1 -11066.003,E2 -11066.003} C_VEL
LIN {X 0,Y 403.19,Z 428.678,A -85,B 0,C 180,E1 -11067.002,E2 -11067.002} C_VEL
LIN {X 0,Y 402.983,Z 430.285,A -85,B 0,C 180,E1 -11069.001,E2 -11069.001} C_VEL
LIN {X 0,Y 402.975,Z 430.519,A -85,B 0,C 180,E1 -11070,E2 -11070} C_VEL
LIN {X 0,Y 403.063,Z 429.746,A -85,B 0,C 180,E1 -11071.998,E2 -11071.998} C_VEL
LIN {X 0,Y 403.189,Z 428.781,A -85,B 0,C 180,E1 -11072.998,E2 -11072.998} C_VEL
LIN {X 0,Y 403.302,Z 427.426,A -85,B 0,C 180,E1 -11073.997,E2 -11073.997} C_VEL
LIN {X 0,Y 403.315,Z 424.586,A -85,B 0,C 180,E1 -11075.5,E2 -11075.5} C_VEL
LIN {X 0,Y 403.727,Z 420.283,A -85,B 0,C 180,E1 -11077.138,E2 -11077.138} C_VEL
LIN {X 0,Y 404.044,Z 415.692,A -85,B 0,C 180,E1 -11078.502,E2 -11078.502} C_VEL
LIN {X 0,Y 404.251,Z 413.42,A -85,B 0,C 180,E1 -11079.078,E2 -11079.078} C_VEL
LIN {X 0,Y 403.83,Z 410.441,A -85,B 0,C 180,E1 -11079.798,E2 -11079.798} C_VEL
LIN {X 0,Y 401.507,Z 405.28,A -85,B 0,C 180,E1 -11080.959,E2 -11080.959} C_VEL
LIN {X 0,Y 399.253,Z 399.568,A -85,B 0,C 180,E1 -11082.072,E2 -11082.072} C_VEL
LIN {X 0,Y 398.939,Z 395.654,A -85,B 0,C 180,E1 -11082.707,E2 -11082.707} C_VEL
LIN {X 0,Y 399.783,Z 386.086,A -85,B 0,C 180,E1 -11083.988,E2 -11083.988} C_VEL
LIN {X 0,Y 400.522,Z 375.007,A -85,B 0,C 180,E1 -11085.183,E2 -11085.183} C_VEL
LIN {X 0,Y 401.287,Z 363.599,A -85,B 0,C 180,E1 -11086.143,E2 -11086.143} C_VEL
LIN {X 0,Y 401.973,Z 351.632,A -85,B 0,C 180,E1 -11086.92,E2 -11086.92} C_VEL
LIN {X 0,Y 401.947,Z 348.295,A -85,B 0,C 180,E1 -11087.103,E2 -11087.103} C_VEL
LIN {X 0,Y 399.17,Z 335.784,A -85,B 0,C 180,E1 -11087.796,E2 -11087.796} C_VEL
LIN {X 0,Y 396.483,Z 325.641,A -85,B 0,C 180,E1 -11088.24,E2 -11088.24} C_VEL
LIN {X 0,Y 396.471,Z 321.078,A -85,B 0,C 180,E1 -11090.765,E2 -11090.765} C_VEL
LIN {X 0,Y 396.533,Z 315.513,A -85,B 0,C 180,E1 -11094.057,E2 -11094.057} C_VEL
LIN {X 0,Y 396.608,Z 309.729,A -85,B 0,C 180,E1 -11097.623,E2 -11097.623} C_VEL
LIN {X 0,Y 396.686,Z 304.512,A -85,B 0,C 180,E1 -11100.917,E2 -11100.917} C_VEL
LIN {X 0,Y 396.979,Z 300.04,A -85,B 0,C 180,E1 -11103.81,E2 -11103.81} C_VEL
LIN {X 0,Y 397.092,Z 300.025,A -85,B 0,C 180,E1 -11107.208,E2 -11107.208} C_VEL
LIN {X 0,Y 397.104,Z 300.022,A -85,B 0,C 180,E1 -11110.445,E2 -11110.445} C_VEL
LIN {X 0,Y 397.103,Z 300.023,A -85,B 0,C 180,E1 -11113.648,E2 -11113.648} C_VEL
LIN {X 0,Y 397.104,Z 300.022,A -85,B 0,C 180,E1 -11116.521,E2 -11116.521} C_VEL
LIN {X 0,Y 397.117,Z 300.02,A -85,B 0,C 180,E1 -11120.423,E2 -11120.423} C_VEL
LIN {X 0,Y 397.089,Z 300.024,A -85,B 0,C 180,E1 -11123.004,E2 -11123.004} C_VEL
LIN {X 0,Y 396.88,Z 300.05,A -85,B 0,C 180,E1 -11126.334,E2 -11126.334} C_VEL
LIN {X 0,Y 396.79,Z 300.253,A -85,B 0,C 180,E1 -11127.15,E2 -11127.15} C_VEL
LIN {X 0,Y 396.587,Z 305.379,A -85,B 0,C 180,E1 -11130.267,E2 -11130.267} C_VEL
LIN {X 0,Y 396.479,Z 310.987,A -85,B 0,C 180,E1 -11133.695,E2 -11133.695} C_VEL
LIN {X 0,Y 396.452,Z 316.68,A -85,B 0,C 180,E1 -11137.194,E2 -11137.194} C_VEL
LIN {X 0,Y 396.387,Z 321.85,A -85,B 0,C 180,E1 -11140.313,E2 -11140.313} C_VEL
LIN {X 0,Y 396.33,Z 325.847,A -85,B 0,C 180,E1 -11142.699,E2 -11142.699} C_VEL
LIN {X 0,Y 399.158,Z 339.292,A -85,B 0,C 180,E1 -11143.292,E2 -11143.292} C_VEL
LIN {X 0,Y 400.614,Z 347.795,A -85,B 0,C 180,E1 -11143.764,E2 -11143.764} C_VEL
LIN {X 0,Y 399.93,Z 360.828,A -85,B 0,C 180,E1 -11144.586,E2 -11144.586} C_VEL
LIN {X 0,Y 399.259,Z 373.076,A -85,B 0,C 180,E1 -11145.588,E2 -11145.588} C_VEL
LIN {X 0,Y 398.691,Z 384.285,A -85,B 0,C 180,E1 -11146.752,E2 -11146.752} C_VEL
LIN {X 0,Y 398,Z 394.267,A -85,B 0,C 180,E1 -11148.025,E2 -11148.025} C_VEL
LIN {X 0,Y 397.431,Z 403.905,A -85,B 0,C 180,E1 -11149.557,E2 -11149.557} C_VEL
LIN {X 0,Y 396.904,Z 411.648,A -85,B 0,C 180,E1 -11151.087,E2 -11151.087} C_VEL
LIN {X 0,Y 396.438,Z 418.771,A -85,B 0,C 180,E1 -11152.871,E2 -11152.871} C_VEL
LIN {X 0,Y 396.244,Z 423.475,A -85,B 0,C 180,E1 -11154.402,E2 -11154.402} C_VEL
LIN {X 0,Y 396.184,Z 427.017,A -85,B 0,C 180,E1 -11155.931,E2 -11155.931} C_VEL
LIN {X 0,Y 396.127,Z 428.779,A -85,B 0,C 180,E1 -11156.949,E2 -11156.949} C_VEL
LIN {X 0,Y 395.995,Z 430.139,A -85,B 0,C 180,E1 -11157.966,E2 -11157.966} C_VEL
LIN {X 0,Y 395.931,Z 431.047,A -85,B 0,C 180,E1 -11158.983,E2 -11158.983} C_VEL
LIN {X 0,Y 395.936,Z 431.51,A -85,B 0,C 180,E1 -11160,E2 -11160} C_VEL
LIN {X 0,Y 395.974,Z 431.572,A -85,B 0,C 180,E1 -11161.017,E2 -11161.017} C_VEL
LIN {X 0,Y 396.07,Z 431.193,A -85,B 0,C 180,E1 -11162.034,E2 -11162.034} C_VEL
LIN {X 0,Y 396.184,Z 430.367,A -85,B 0,C 180,E1 -11163.051,E2 -11163.051} C_VEL
LIN {X 0,Y 396.329,Z 429.136,A -85,B 0,C 180,E1 -11164.067,E2 -11164.067} C_VEL
LIN {X 0,Y 396.416,Z 426.456,A -85,B 0,C 180,E1 -11165.596,E2 -11165.596} C_VEL
LIN {X 0,Y 396.858,Z 421.911,A -85,B 0,C 180,E1 -11167.381,E2 -11167.381} C_VEL
LIN {X 0,Y 397.449,Z 415.776,A -85,B 0,C 180,E1 -11169.157,E2 -11169.157} C_VEL
LIN {X 0,Y 398.041,Z 408.955,A -85,B 0,C 180,E1 -11170.684,E2 -11170.684} C_VEL
LIN {X 0,Y 398.757,Z 400.47,A -85,B 0,C 180,E1 -11172.21,E2 -11172.21} C_VEL
LIN {X 0,Y 399.541,Z 391.77,A -85,B 0,C 180,E1 -11173.478,E2 -11173.478} C_VEL
LIN {X 0,Y 400.429,Z 380.931,A -85,B 0,C 180,E1 -11174.758,E2 -11174.758} C_VEL
LIN {X 0,Y 401.154,Z 370.5,A -85,B 0,C 180,E1 -11175.756,E2 -11175.756} C_VEL
LIN {X 0,Y 402.026,Z 357.252,A -85,B 0,C 180,E1 -11176.753,E2 -11176.753} C_VEL
LIN {X 0,Y 402.355,Z 348.655,A -85,B 0,C 180,E1 -11177.274,E2 -11177.274} C_VEL
LIN {X 0,Y 399.541,Z 337.539,A -85,B 0,C 180,E1 -11178.015,E2 -11178.015} C_VEL
LIN {X 0,Y 397.023,Z 329.628,A -85,B 0,C 180,E1 -11178.505,E2 -11178.505} C_VEL
LIN {X 0,Y 397.097,Z 324.043,A -85,B 0,C 180,E1 -11181.819,E2 -11181.819} C_VEL
LIN {X 0,Y 397.196,Z 318.282,A -85,B 0,C 180,E1 -11185.129,E2 -11185.129} C_VEL
LIN {X 0,Y 397.38,Z 312.171,A -85,B 0,C 180,E1 -11188.523,E2 -11188.523} C_VEL
LIN {X 0,Y 397.614,Z 305.623,A -85,B 0,C 180,E1 -11192.023,E2 -11192.023} C_VEL
LIN {X 0,Y 397.47,Z 302.293,A -85,B 0,C 180,E1 -11193.793,E2 -11193.793} C_VEL
LIN {X 0,Y 397.065,Z 300.029,A -85,B 0,C 180,E1 -11195.117,E2 -11195.117} C_VEL
LIN {X 0,Y 397.102,Z 300.022,A -85,B 0,C 180,E1 -11198.275,E2 -11198.275} C_VEL
LIN {X 0,Y 397.088,Z 300.023,A -85,B 0,C 180,E1 -11200.909,E2 -11200.909} C_VEL
LIN {X 0,Y 397.103,Z 300.021,A -85,B 0,C 180,E1 -11204.618,E2 -11204.618} C_VEL
LIN {X 0,Y 397.145,Z 300.297,A -85,B 0,C 180,E1 -11204.939,E2 -11204.939} C_VEL
LIN {X 0,Y 398.67,Z 308.132,A -85,B 0,C 180,E1 -11208.522,E2 -11208.522} C_VEL
LIN {X 0,Y 399.962,Z 314.732,A -85,B 0,C 180,E1 -11211.406,E2 -11211.406} C_VEL
LIN {X 0,Y 400.567,Z 319.466,A -85,B 0,C 180,E1 -11213.378,E2 -11213.378} C_VEL
LIN {X 0,Y 400.019,Z 325.663,A -85,B 0,C 180,E1 -11215.791,E2 -11215.791} C_VEL
LIN {X 0,Y 399.239,Z 334.916,A -85,B 0,C 180,E1 -11219.303,E2 -11219.303} C_VEL
LIN {X 0,Y 398.325,Z 345.694,A -85,B 0,C 180,E1 -11223.261,E2 -11223.261} C_VEL
LIN {X 0,Y 397.734,Z 354.593,A -85,B 0,C 180,E1 -11226.458,E2 -11226.458} C_VEL
LIN {X 0,Y 397.206,Z 363.717,A -85,B 0,C 180,E1 -11229.679,E2 -11229.679} C_VEL
LIN {X 0,Y 396.873,Z 369.556,A -85,B 0,C 180,E1 -11231.714,E2 -11231.714} C_VEL
LIN {X 0,Y 399.203,Z 385.445,A -85,B 0,C 180,E1 -11232.387,E2 -11232.387} C_VEL
LIN {X 0,Y 400.824,Z 398.481,A -85,B 0,C 180,E1 -11233.139,E2 -11233.139} C_VEL
LIN {X 0,Y 400.756,Z 405.19,A -85,B 0,C 180,E1 -11233.578,E2 -11233.578} C_VEL
LIN {X 0,Y 399.895,Z 416.469,A -85,B 0,C 180,E1 -11234.454,E2 -11234.454} C_VEL
LIN {X 0,Y 398.943,Z 428.011,A -85,B 0,C 180,E1 -11235.591,E2 -11235.591} C_VEL
LIN {X 0,Y 398.259,Z 437.417,A -85,B 0,C 180,E1 -11236.738,E2 -11236.738} C_VEL
LIN {X 0,Y 397.528,Z 446.051,A -85,B 0,C 180,E1 -11238.011,E2 -11238.011} C_VEL
LIN {X 0,Y 396.884,Z 454.476,A -85,B 0,C 180,E1 -11239.542,E2 -11239.542} C_VEL
LIN {X 0,Y 396.451,Z 461.27,A -85,B 0,C 180,E1 -11241.077,E2 -11241.077} C_VEL
LIN {X 0,Y 396.099,Z 467.511,A -85,B 0,C 180,E1 -11242.865,E2 -11242.865} C_VEL
LIN {X 0,Y 395.991,Z 471.563,A -85,B 0,C 180,E1 -11244.398,E2 -11244.398} C_VEL
LIN {X 0,Y 395.835,Z 474.53,A -85,B 0,C 180,E1 -11245.927,E2 -11245.927} C_VEL
LIN {X 0,Y 395.935,Z 475.964,A -85,B 0,C 180,E1 -11246.947,E2 -11246.947} C_VEL
LIN {X 0,Y 395.975,Z 477.548,A -85,B 0,C 180,E1 -11248.983,E2 -11248.983} C_VEL
LIN {X 0,Y 395.968,Z 477.729,A -85,B 0,C 180,E1 -11250,E2 -11250} C_VEL
LIN {X 0,Y 395.979,Z 477.473,A -85,B 0,C 180,E1 -11251.017,E2 -11251.017} C_VEL
LIN {X 0,Y 395.942,Z 475.711,A -85,B 0,C 180,E1 -11253.052,E2 -11253.052} C_VEL
LIN {X 0,Y 395.855,Z 474.2,A -85,B 0,C 180,E1 -11254.072,E2 -11254.072} C_VEL
LIN {X 0,Y 396.015,Z 471.087,A -85,B 0,C 180,E1 -11255.601,E2 -11255.601} C_VEL
LIN {X 0,Y 396.099,Z 466.878,A -85,B 0,C 180,E1 -11257.135,E2 -11257.135} C_VEL
LIN {X 0,Y 396.457,Z 460.572,A -85,B 0,C 180,E1 -11258.923,E2 -11258.923} C_VEL
LIN {X 0,Y 396.852,Z 453.694,A -85,B 0,C 180,E1 -11260.458,E2 -11260.458} C_VEL
LIN {X 0,Y 397.407,Z 446.662,A -85,B 0,C 180,E1 -11261.734,E2 -11261.734} C_VEL
LIN {X 0,Y 398.039,Z 438.163,A -85,B 0,C 180,E1 -11263.01,E2 -11263.01} C_VEL
LIN {X 0,Y 398.783,Z 428.013,A -85,B 0,C 180,E1 -11264.284,E2 -11264.284} C_VEL
LIN {X 0,Y 399.653,Z 416.806,A -85,B 0,C 180,E1 -11265.425,E2 -11265.425} C_VEL
LIN {X 0,Y 400.705,Z 404.415,A -85,B 0,C 180,E1 -11266.429,E2 -11266.429} C_VEL
LIN {X 0,Y 400.865,Z 398.871,A -85,B 0,C 180,E1 -11266.815,E2 -11266.815} C_VEL
LIN {X 0,Y 399.462,Z 386.127,A -85,B 0,C 180,E1 -11267.627,E2 -11267.627} C_VEL
LIN {X 0,Y 397.859,Z 372.596,A -85,B 0,C 180,E1 -11268.297,E2 -11268.297} C_VEL
LIN {X 0,Y 396.789,Z 366.099,A -85,B 0,C 180,E1 -11268.592,E2 -11268.592} C_VEL
LIN {X 0,Y 397.297,Z 355.109,A -85,B 0,C 180,E1 -11272.354,E2 -11272.354} C_VEL
LIN {X 0,Y 397.839,Z 345.63,A -85,B 0,C 180,E1 -11275.718,E2 -11275.718} C_VEL
LIN {X 0,Y 398.448,Z 336.769,A -85,B 0,C 180,E1 -11279.016,E2 -11279.016} C_VEL
LIN {X 0,Y 399.245,Z 328.405,A -85,B 0,C 180,E1 -11282.333,E2 -11282.333} C_VEL
LIN {X 0,Y 400.141,Z 321.246,A -85,B 0,C 180,E1 -11285.423,E2 -11285.423} C_VEL
LIN {X 0,Y 400.389,Z 317.556,A -85,B 0,C 180,E1 -11287.202,E2 -11287.202} C_VEL
LIN {X 0,Y 399.567,Z 312.77,A -85,B 0,C 180,E1 -11289.941,E2 -11289.941} C_VEL
LIN {X 0,Y 398.947,Z 309.362,A -85,B 0,C 180,E1 -11292.278,E2 -11292.278} C_VEL
LIN {X 0,Y 398.312,Z 306.096,A -85,B 0,C 180,E1 -11295.107,E2 -11295.107} C_VEL
LIN {X 0,Y 397.841,Z 303.82,A -85,B 0,C 180,E1 -11297.898,E2 -11297.898} C_VEL
LIN {X 0,Y 397.55,Z 302.278,A -85,B 0,C 180,E1 -11301.064,E2 -11301.064} C_VEL
LIN {X 0,Y 397.429,Z 301.727,A -85,B 0,C 180,E1 -11304.435,E2 -11304.435} C_VEL
LIN {X 0,Y 397.447,Z 301.908,A -85,B 0,C 180,E1 -11306.758,E2 -11306.758} C_VEL
LIN {X 0,Y 397.604,Z 302.805,A -85,B 0,C 180,E1 -11310.335,E2 -11310.335} C_VEL
LIN {X 0,Y 397.762,Z 303.719,A -85,B 0,C 180,E1 -11312.652,E2 -11312.652} C_VEL
LIN {X 0,Y 397.814,Z 304.835,A -85,B 0,C 180,E1 -11314.913,E2 -11314.913} C_VEL
LIN {X 0,Y 397.789,Z 306.096,A -85,B 0,C 180,E1 -11317.127,E2 -11317.127} C_VEL
LIN {X 0,Y 397.642,Z 308.197,A -85,B 0,C 180,E1 -11320.378,E2 -11320.378} C_VEL
LIN {X 0,Y 397.56,Z 309.131,A -85,B 0,C 180,E1 -11321.627,E2 -11321.627} C_VEL
LIN {X 0,Y 402.204,Z 321.791,A -85,B 0,C 180,E1 -11322.526,E2 -11322.526} C_VEL
LIN {X 0,Y 403.138,Z 324.917,A -85,B 0,C 180,E1 -11322.761,E2 -11322.761} C_VEL
LIN {X 0,Y 402.436,Z 338.627,A -85,B 0,C 180,E1 -11323.644,E2 -11323.644} C_VEL
LIN {X 0,Y 401.547,Z 350.906,A -85,B 0,C 180,E1 -11324.678,E2 -11324.678} C_VEL
LIN {X 0,Y 400.763,Z 361.434,A -85,B 0,C 180,E1 -11325.788,E2 -11325.788} C_VEL
LIN {X 0,Y 399.933,Z 371.115,A -85,B 0,C 180,E1 -11327.053,E2 -11327.053} C_VEL
LIN {X 0,Y 399.151,Z 380.462,A -85,B 0,C 180,E1 -11328.575,E2 -11328.575} C_VEL
LIN {X 0,Y 398.359,Z 387.94,A -85,B 0,C 180,E1 -11330.095,E2 -11330.095} C_VEL
LIN {X 0,Y 397.693,Z 394.771,A -85,B 0,C 180,E1 -11331.873,E2 -11331.873} C_VEL
LIN {X 0,Y 397.167,Z 399.256,A -85,B 0,C 180,E1 -11333.395,E2 -11333.395} C_VEL
LIN {X 0,Y 396.986,Z 402.571,A -85,B 0,C 180,E1 -11334.922,E2 -11334.922} C_VEL
LIN {X 0,Y 396.721,Z 404.218,A -85,B 0,C 180,E1 -11335.937,E2 -11335.937} C_VEL
LIN {X 0,Y 396.436,Z 405.423,A -85,B 0,C 180,E1 -11336.951,E2 -11336.951} C_VEL
LIN {X 0,Y 396.248,Z 406.216,A -85,B 0,C 180,E1 -11337.967,E2 -11337.967} C_VEL
LIN {X 0,Y 396.159,Z 406.584,A -85,B 0,C 180,E1 -11338.984,E2 -11338.984} C_VEL
LIN {X 0,Y 396.12,Z 406.498,A -85,B 0,C 180,E1 -11340,E2 -11340} C_VEL
LIN {X 0,Y 396.131,Z 406.006,A -85,B 0,C 180,E1 -11341.017,E2 -11341.017} C_VEL
LIN {X 0,Y 396.222,Z 405.106,A -85,B 0,C 180,E1 -11342.033,E2 -11342.033} C_VEL
LIN {X 0,Y 396.418,Z 403.742,A -85,B 0,C 180,E1 -11343.049,E2 -11343.049} C_VEL
LIN {X 0,Y 396.619,Z 400.901,A -85,B 0,C 180,E1 -11344.574,E2 -11344.574} C_VEL
LIN {X 0,Y 396.651,Z 397.017,A -85,B 0,C 180,E1 -11346.103,E2 -11346.103} C_VEL
LIN {X 0,Y 397.022,Z 391.309,A -85,B 0,C 180,E1 -11347.802,E2 -11347.802} C_VEL
LIN {X 0,Y 397.437,Z 384.401,A -85,B 0,C 180,E1 -11349.414,E2 -11349.414} C_VEL
LIN {X 0,Y 397.963,Z 376.156,A -85,B 0,C 180,E1 -11350.944,E2 -11350.944} C_VEL
LIN {X 0,Y 398.497,Z 367.777,A -85,B 0,C 180,E1 -11352.218,E2 -11352.218} C_VEL
LIN {X 0,Y 399.184,Z 357.612,A -85,B 0,C 180,E1 -11353.49,E2 -11353.49} C_VEL
LIN {X 0,Y 399.787,Z 345.842,A -85,B 0,C 180,E1 -11354.671,E2 -11354.671} C_VEL
LIN {X 0,Y 400.358,Z 333.462,A -85,B 0,C 180,E1 -11355.658,E2 -11355.658} C_VEL
LIN {X 0,Y 400.922,Z 321.137,A -85,B 0,C 180,E1 -11356.407,E2 -11356.407} C_VEL
LIN {X 0,Y 397.987,Z 308.056,A -85,B 0,C 180,E1 -11357.115,E2 -11357.115} C_VEL
LIN {X 0,Y 396.402,Z 301.328,A -85,B 0,C 180,E1 -11357.423,E2 -11357.423} C_VEL
LIN {X 0,Y 396.38,Z 300.114,A -85,B 0,C 180,E1 -11358.612,E2 -11358.612} C_VEL
LIN {X 0,Y 396.651,Z 300.074,A -85,B 0,C 180,E1 -11360.755,E2 -11360.755} C_VEL
LIN {X 0,Y 396.96,Z 300.04,A -85,B 0,C 180,E1 -11364.03,E2 -11364.03} C_VEL
LIN {X 0,Y 397.179,Z 300.006,A -85,B 0,C 180,E1 -11367.391,E2 -11367.391} C_VEL
LIN {X 0,Y 397.081,Z 300.017,A -85,B 0,C 180,E1 -11370.882,E2 -11370.882} C_VEL
LIN {X 0,Y 397.128,Z 300.015,A -85,B 0,C 180,E1 -11374.493,E2 -11374.493} C_VEL
LIN {X 0,Y 397.105,Z 300.021,A -85,B 0,C 180,E1 -11378.275,E2 -11378.275} C_VEL
LIN {X 0,Y 397.091,Z 300.022,A -85,B 0,C 180,E1 -11380.909,E2 -11380.909} C_VEL
LIN {X 0,Y 397.105,Z 300.023,A -85,B 0,C 180,E1 -11383.648,E2 -11383.648} C_VEL
LIN {X 0,Y 397.105,Z 300.017,A -85,B 0,C 180,E1 -11386.521,E2 -11386.521} C_VEL
LIN {X 0,Y 397.116,Z 300.018,A -85,B 0,C 180,E1 -11390.423,E2 -11390.423} C_VEL
LIN {X 0,Y 397.097,Z 300.021,A -85,B 0,C 180,E1 -11393.005,E2 -11393.005} C_VEL
LIN {X 0,Y 396.942,Z 300.207,A -85,B 0,C 180,E1 -11396.512,E2 -11396.512} C_VEL
LIN {X 0,Y 396.667,Z 306.208,A -85,B 0,C 180,E1 -11400.258,E2 -11400.258} C_VEL
LIN {X 0,Y 396.571,Z 311.683,A -85,B 0,C 180,E1 -11403.701,E2 -11403.701} C_VEL
LIN {X 0,Y 396.527,Z 317.357,A -85,B 0,C 180,E1 -11407.168,E2 -11407.168} C_VEL
LIN {X 0,Y 396.514,Z 322.804,A -85,B 0,C 180,E1 -11410.32,E2 -11410.32} C_VEL
LIN {X 0,Y 396.468,Z 325.726,A -85,B 0,C 180,E1 -11411.875,E2 -11411.875} C_VEL
LIN {X 0,Y 399.989,Z 339.242,A -85,B 0,C 180,E1 -11412.476,E2 -11412.476} C_VEL
LIN {X 0,Y 401.956,Z 348.884,A -85,B 0,C 180,E1 -11413.026,E2 -11413.026} C_VEL
LIN {X 0,Y 401.488,Z 360.554,A -85,B 0,C 180,E1 -11413.735,E2 -11413.735} C_VEL
LIN {X 0,Y 400.777,Z 371.784,A -85,B 0,C 180,E1 -11414.619,E2 -11414.619} C_VEL
LIN {X 0,Y 399.982,Z 383.092,A -85,B 0,C 180,E1 -11415.76,E2 -11415.76} C_VEL
LIN {X 0,Y 399.12,Z 393.172,A -85,B 0,C 180,E1 -11417.026,E2 -11417.026} C_VEL
LIN {X 0,Y 398.296,Z 402.787,A -85,B 0,C 180,E1 -11418.55,E2 -11418.55} C_VEL
LIN {X 0,Y 397.567,Z 410.516,A -85,B 0,C 180,E1 -11420.075,E2 -11420.075} C_VEL
LIN {X 0,Y 397.083,Z 415.734,A -85,B 0,C 180,E1 -11421.347,E2 -11421.347} C_VEL
LIN {X 0,Y 396.672,Z 420.831,A -85,B 0,C 180,E1 -11422.876,E2 -11422.876} C_VEL
LIN {X 0,Y 396.29,Z 424.781,A -85,B 0,C 180,E1 -11424.402,E2 -11424.402} C_VEL
LIN {X 0,Y 396.24,Z 427.681,A -85,B 0,C 180,E1 -11425.932,E2 -11425.932} C_VEL
LIN {X 0,Y 396.131,Z 429.092,A -85,B 0,C 180,E1 -11426.949,E2 -11426.949} C_VEL
LIN {X 0,Y 395.907,Z 430.7,A -85,B 0,C 180,E1 -11428.983,E2 -11428.983} C_VEL
LIN {X 0,Y 395.896,Z 430.934,A -85,B 0,C 180,E1 -11430,E2 -11430} C_VEL
LIN {X 0,Y 395.994,Z 430.159,A -85,B 0,C 180,E1 -11432.034,E2 -11432.034} C_VEL
LIN {X 0,Y 396.129,Z 429.194,A -85,B 0,C 180,E1 -11433.051,E2 -11433.051} C_VEL
LIN {X 0,Y 396.229,Z 427.84,A -85,B 0,C 180,E1 -11434.069,E2 -11434.069} C_VEL
LIN {X 0,Y 396.273,Z 424.998,A -85,B 0,C 180,E1 -11435.598,E2 -11435.598} C_VEL
LIN {X 0,Y 396.677,Z 420.968,A -85,B 0,C 180,E1 -11437.176,E2 -11437.176} C_VEL
LIN {X 0,Y 397.047,Z 416.102,A -85,B 0,C 180,E1 -11438.653,E2 -11438.653} C_VEL
LIN {X 0,Y 397.672,Z 409.762,A -85,B 0,C 180,E1 -11440.179,E2 -11440.179} C_VEL
LIN {X 0,Y 398.342,Z 401.887,A -85,B 0,C 180,E1 -11441.706,E2 -11441.706} C_VEL
LIN {X 0,Y 398.939,Z 395.654,A -85,B 0,C 180,E1 -11442.707,E2 -11442.707} C_VEL
LIN {X 0,Y 398.621,Z 391.585,A -85,B 0,C 180,E1 -11443.319,E2 -11443.319} C_VEL
LIN {X 0,Y 396.395,Z 384.748,A -85,B 0,C 180,E1 -11444.303,E2 -11444.303} C_VEL
LIN {X 0,Y 394.192,Z 377.459,A -85,B 0,C 180,E1 -11445.219,E2 -11445.219} C_VEL
LIN {X 0,Y 393.905,Z 372.587,A -85,B 0,C 180,E1 -11445.716,E2 -11445.716} C_VEL
LIN {X 0,Y 394.666,Z 362.288,A -85,B 0,C 180,E1 -11446.554,E2 -11446.554} C_VEL
LIN {X 0,Y 395.227,Z 351.067,A -85,B 0,C 180,E1 -11447.272,E2 -11447.272} C_VEL
LIN {X 0,Y 393.755,Z 342.741,A -85,B 0,C 180,E1 -11447.771,E2 -11447.771} C_VEL
LIN {X 0,Y 390.527,Z 330.026,A -85,B 0,C 180,E1 -11448.407,E2 -11448.407} C_VEL
LIN {X 0,Y 389.449,Z 326.027,A -85,B 0,C 180,E1 -11448.57,E2 -11448.57} C_VEL
LIN {X 0,Y 389.44,Z 321.372,A -85,B 0,C 180,E1 -11451.157,E2 -11451.157} C_VEL
LIN {X 0,Y 389.5,Z 315.716,A -85,B 0,C 180,E1 -11454.52,E2 -11454.52} C_VEL
LIN {X 0,Y 389.562,Z 310.148,A -85,B 0,C 180,E1 -11457.973,E2 -11457.973} C_VEL
LIN {X 0,Y 389.676,Z 304.53,A -85,B 0,C 180,E1 -11461.536,E2 -11461.536} C_VEL
LIN {X 0,Y 389.937,Z 300.918,A -85,B 0,C 180,E1 -11463.812,E2 -11463.812} C_VEL
LIN {X 0,Y 390.033,Z 300.903,A -85,B 0,C 180,E1 -11466.486,E2 -11466.486} C_VEL
LIN {X 0,Y 390.071,Z 300.897,A -85,B 0,C 180,E1 -11469.218,E2 -11469.218} C_VEL
LIN {X 0,Y 390.045,Z 300.903,A -85,B 0,C 180,E1 -11472.374,E2 -11472.374} C_VEL
LIN {X 0,Y 390.047,Z 300.901,A -85,B 0,C 180,E1 -11475.354,E2 -11475.354} C_VEL
LIN {X 0,Y 390.034,Z 300.901,A -85,B 0,C 180,E1 -11478.187,E2 -11478.187} C_VEL
LIN {X 0,Y 390.093,Z 300.893,A -85,B 0,C 180,E1 -11480.908,E2 -11480.908} C_VEL
LIN {X 0,Y 389.977,Z 300.908,A -85,B 0,C 180,E1 -11484.191,E2 -11484.191} C_VEL
LIN {X 0,Y 389.744,Z 301.04,A -85,B 0,C 180,E1 -11487.096,E2 -11487.096} C_VEL
LIN {X 0,Y 389.485,Z 307.154,A -85,B 0,C 180,E1 -11490.843,E2 -11490.843} C_VEL
LIN {X 0,Y 389.432,Z 313.064,A -85,B 0,C 180,E1 -11494.468,E2 -11494.468} C_VEL
LIN {X 0,Y 389.363,Z 318.329,A -85,B 0,C 180,E1 -11497.725,E2 -11497.725} C_VEL
LIN {X 0,Y 389.274,Z 323.824,A -85,B 0,C 180,E1 -11501.036,E2 -11501.036} C_VEL
LIN {X 0,Y 389.28,Z 326.309,A -85,B 0,C 180,E1 -11502.47,E2 -11502.47} C_VEL
LIN {X 0,Y 391.961,Z 339.067,A -85,B 0,C 180,E1 -11503.041,E2 -11503.041} C_VEL
LIN {X 0,Y 393.627,Z 348.892,A -85,B 0,C 180,E1 -11503.601,E2 -11503.601} C_VEL
LIN {X 0,Y 392.946,Z 361.74,A -85,B 0,C 180,E1 -11504.438,E2 -11504.438} C_VEL
LIN {X 0,Y 392.254,Z 374.016,A -85,B 0,C 180,E1 -11505.473,E2 -11505.473} C_VEL
LIN {X 0,Y 391.68,Z 385.014,A -85,B 0,C 180,E1 -11506.643,E2 -11506.643} C_VEL
LIN {X 0,Y 391.01,Z 394.048,A -85,B 0,C 180,E1 -11507.808,E2 -11507.808} C_VEL
LIN {X 0,Y 390.412,Z 403.813,A -85,B 0,C 180,E1 -11509.367,E2 -11509.367} C_VEL
LIN {X 0,Y 389.868,Z 411.694,A -85,B 0,C 180,E1 -11510.925,E2 -11510.925} C_VEL
LIN {X 0,Y 389.401,Z 418.904,A -85,B 0,C 180,E1 -11512.742,E2 -11512.742} C_VEL
LIN {X 0,Y 389.196,Z 423.697,A -85,B 0,C 180,E1 -11514.3,E2 -11514.3} C_VEL
LIN {X 0,Y 389.095,Z 427.319,A -85,B 0,C 180,E1 -11515.857,E2 -11515.857} C_VEL
LIN {X 0,Y 389.067,Z 429.118,A -85,B 0,C 180,E1 -11516.893,E2 -11516.893} C_VEL
LIN {X 0,Y 388.928,Z 430.508,A -85,B 0,C 180,E1 -11517.929,E2 -11517.929} C_VEL
LIN {X 0,Y 388.857,Z 431.466,A -85,B 0,C 180,E1 -11518.964,E2 -11518.964} C_VEL
LIN {X 0,Y 388.858,Z 431.958,A -85,B 0,C 180,E1 -11520,E2 -11520} C_VEL
LIN {X 0,Y 388.898,Z 432.047,A -85,B 0,C 180,E1 -11521.035,E2 -11521.035} C_VEL
LIN {X 0,Y 388.999,Z 431.717,A -85,B 0,C 180,E1 -11522.071,E2 -11522.071} C_VEL
LIN {X 0,Y 389.125,Z 430.921,A -85,B 0,C 180,E1 -11523.106,E2 -11523.106} C_VEL
LIN {X 0,Y 389.286,Z 429.717,A -85,B 0,C 180,E1 -11524.141,E2 -11524.141} C_VEL
LIN {X 0,Y 389.381,Z 427.082,A -85,B 0,C 180,E1 -11525.697,E2 -11525.697} C_VEL
LIN {X 0,Y 389.862,Z 422.689,A -85,B 0,C 180,E1 -11527.483,E2 -11527.483} C_VEL
LIN {X 0,Y 390.494,Z 416.521,A -85,B 0,C 180,E1 -11529.322,E2 -11529.322} C_VEL
LIN {X 0,Y 391.114,Z 409.815,A -85,B 0,C 180,E1 -11530.876,E2 -11530.876} C_VEL
LIN {X 0,Y 391.886,Z 401.407,A -85,B 0,C 180,E1 -11532.428,E2 -11532.428} C_VEL
LIN {X 0,Y 392.709,Z 392.803,A -85,B 0,C 180,E1 -11533.717,E2 -11533.717} C_VEL
LIN {X 0,Y 393.67,Z 382.033,A -85,B 0,C 180,E1 -11535.025,E2 -11535.025} C_VEL
LIN {X 0,Y 394.457,Z 371.923,A -85,B 0,C 180,E1 -11536.031,E2 -11536.031} C_VEL
LIN {X 0,Y 395.363,Z 358.829,A -85,B 0,C 180,E1 -11537.056,E2 -11537.056} C_VEL
LIN {X 0,Y 395.852,Z 350.66,A -85,B 0,C 180,E1 -11537.567,E2 -11537.567} C_VEL
LIN {X 0,Y 392.931,Z 338.878,A -85,B 0,C 180,E1 -11538.396,E2 -11538.396} C_VEL
LIN {X 0,Y 390.049,Z 330.177,A -85,B 0,C 180,E1 -11538.993,E2 -11538.993} C_VEL
LIN {X 0,Y 390.133,Z 324.758,A -85,B 0,C 180,E1 -11542.229,E2 -11542.229} C_VEL
LIN {X 0,Y 390.266,Z 318.977,A -85,B 0,C 180,E1 -11545.607,E2 -11545.607} C_VEL
LIN {X 0,Y 390.534,Z 312.845,A -85,B 0,C 180,E1 -11549.071,E2 -11549.071} C_VEL
LIN {X 0,Y 390.788,Z 306.3,A -85,B 0,C 180,E1 -11552.651,E2 -11552.651} C_VEL
LIN {X 0,Y 390.536,Z 303.639,A -85,B 0,C 180,E1 -11554.126,E2 -11554.126} C_VEL
LIN {X 0,Y 390.039,Z 300.903,A -85,B 0,C 180,E1 -11555.731,E2 -11555.731} C_VEL
LIN {X 0,Y 390.069,Z 300.898,A -85,B 0,C 180,E1 -11559.218,E2 -11559.218} C_VEL
LIN {X 0,Y 390.041,Z 300.901,A -85,B 0,C 180,E1 -11562.373,E2 -11562.373} C_VEL
LIN {X 0,Y 390.084,Z 301.097,A -85,B 0,C 180,E1 -11564.534,E2 -11564.534} C_VEL
LIN {X 0,Y 391.468,Z 308.317,A -85,B 0,C 180,E1 -11567.915,E2 -11567.915} C_VEL
LIN {X 0,Y 392.962,Z 315.78,A -85,B 0,C 180,E1 -11571.247,E2 -11571.247} C_VEL
LIN {X 0,Y 393.567,Z 321.048,A -85,B 0,C 180,E1 -11573.473,E2 -11573.473} C_VEL
LIN {X 0,Y 392.765,Z 329.63,A -85,B 0,C 180,E1 -11576.851,E2 -11576.851} C_VEL
LIN {X 0,Y 391.909,Z 339.055,A -85,B 0,C 180,E1 -11580.452,E2 -11580.452} C_VEL
LIN {X 0,Y 391.067,Z 349.811,A -85,B 0,C 180,E1 -11584.449,E2 -11584.449} C_VEL
LIN {X 0,Y 390.419,Z 359.004,A -85,B 0,C 180,E1 -11587.789,E2 -11587.789} C_VEL
LIN {X 0,Y 389.87,Z 368.159,A -85,B 0,C 180,E1 -11591.066,E2 -11591.066} C_VEL
LIN {X 0,Y 389.83,Z 369.114,A -85,B 0,C 180,E1 -11591.405,E2 -11591.405} C_VEL
LIN {X 0,Y 392.071,Z 384.383,A -85,B 0,C 180,E1 -11592.056,E2 -11592.056} C_VEL
LIN {X 0,Y 393.65,Z 397.102,A -85,B 0,C 180,E1 -11592.794,E2 -11592.794} C_VEL
LIN {X 0,Y 394.005,Z 402.723,A -85,B 0,C 180,E1 -11593.175,E2 -11593.175} C_VEL
LIN {X 0,Y 393.119,Z 414.175,A -85,B 0,C 180,E1 -11594.046,E2 -11594.046} C_VEL
LIN {X 0,Y 392.204,Z 424.924,A -85,B 0,C 180,E1 -11595.073,E2 -11595.073} C_VEL
LIN {X 0,Y 391.447,Z 435.194,A -85,B 0,C 180,E1 -11596.3,E2 -11596.3} C_VEL
LIN {X 0,Y 390.555,Z 445.331,A -85,B 0,C 180,E1 -11597.793,E2 -11597.793} C_VEL
LIN {X 0,Y 389.83,Z 453.787,A -85,B 0,C 180,E1 -11599.351,E2 -11599.351} C_VEL
LIN {X 0,Y 389.395,Z 460.601,A -85,B 0,C 180,E1 -11600.914,E2 -11600.914} C_VEL
LIN {X 0,Y 389.029,Z 466.86,A -85,B 0,C 180,E1 -11602.735,E2 -11602.735} C_VEL
LIN {X 0,Y 388.919,Z 470.928,A -85,B 0,C 180,E1 -11604.296,E2 -11604.296} C_VEL
LIN {X 0,Y 388.763,Z 473.907,A -85,B 0,C 180,E1 -11605.853,E2 -11605.853} C_VEL
LIN {X 0,Y 388.856,Z 475.354,A -85,B 0,C 180,E1 -11606.892,E2 -11606.892} C_VEL
LIN {X 0,Y 388.909,Z 476.946,A -85,B 0,C 180,E1 -11608.965,E2 -11608.965} C_VEL
LIN {X 0,Y 388.902,Z 477.176,A -85,B 0,C 180,E1 -11610,E2 -11610} C_VEL
LIN {X 0,Y 388.898,Z 476.963,A -85,B 0,C 180,E1 -11611.035,E2 -11611.035} C_VEL
LIN {X 0,Y 388.856,Z 476.341,A -85,B 0,C 180,E1 -11612.072,E2 -11612.072} C_VEL
LIN {X 0,Y 388.839,Z 475.301,A -85,B 0,C 180,E1 -11613.108,E2 -11613.108} C_VEL
LIN {X 0,Y 388.781,Z 473.775,A -85,B 0,C 180,E1 -11614.147,E2 -11614.147} C_VEL
LIN {X 0,Y 388.913,Z 470.658,A -85,B 0,C 180,E1 -11615.704,E2 -11615.704} C_VEL
LIN {X 0,Y 389.029,Z 466.457,A -85,B 0,C 180,E1 -11617.265,E2 -11617.265} C_VEL
LIN {X 0,Y 389.398,Z 460.155,A -85,B 0,C 180,E1 -11619.086,E2 -11619.086} C_VEL
LIN {X 0,Y 389.829,Z 453.278,A -85,B 0,C 180,E1 -11620.649,E2 -11620.649} C_VEL
LIN {X 0,Y 390.422,Z 446.248,A -85,B 0,C 180,E1 -11621.947,E2 -11621.947} C_VEL
LIN {X 0,Y 391.101,Z 437.748,A -85,B 0,C 180,E1 -11623.245,E2 -11623.245} C_VEL
LIN {X 0,Y 391.96,Z 426.453,A -85,B 0,C 180,E1 -11624.671,E2 -11624.671} C_VEL
LIN {X 0,Y 392.933,Z 415.126,A -85,B 0,C 180,E1 -11625.829,E2 -11625.829} C_VEL
LIN {X 0,Y 394.012,Z 402.593,A -85,B 0,C 180,E1 -11626.849,E2 -11626.849} C_VEL
LIN {X 0,Y 393.532,Z 395.938,A -85,B 0,C 180,E1 -11627.339,E2 -11627.339} C_VEL
LIN {X 0,Y 392.332,Z 382.916,A -85,B 0,C 180,E1 -11628.154,E2 -11628.154} C_VEL
LIN {X 0,Y 390.904,Z 372.079,A -85,B 0,C 180,E1 -11628.712,E2 -11628.712} C_VEL
LIN {X 0,Y 389.764,Z 365.252,A -85,B 0,C 180,E1 -11629.042,E2 -11629.042} C_VEL
LIN {X 0,Y 390.3,Z 354.641,A -85,B 0,C 180,E1 -11632.777,E2 -11632.777} C_VEL
LIN {X 0,Y 390.823,Z 345.924,A -85,B 0,C 180,E1 -11635.956,E2 -11635.956} C_VEL
LIN {X 0,Y 391.564,Z 336.496,A -85,B 0,C 180,E1 -11639.577,E2 -11639.577} C_VEL
LIN {X 0,Y 392.333,Z 329.011,A -85,B 0,C 180,E1 -11642.656,E2 -11642.656} C_VEL
LIN {X 0,Y 393.373,Z 321.316,A -85,B 0,C 180,E1 -11646.127,E2 -11646.127} C_VEL
LIN {X 0,Y 393.434,Z 318.817,A -85,B 0,C 180,E1 -11647.398,E2 -11647.398} C_VEL
LIN {X 0,Y 392.663,Z 314.247,A -85,B 0,C 180,E1 -11650.116,E2 -11650.116} C_VEL
LIN {X 0,Y 391.892,Z 310.338,A -85,B 0,C 180,E1 -11652.959,E2 -11652.959} C_VEL
LIN {X 0,Y 391.305,Z 307.229,A -85,B 0,C 180,E1 -11655.924,E2 -11655.924} C_VEL
LIN {X 0,Y 390.87,Z 305.024,A -85,B 0,C 180,E1 -11659.041,E2 -11659.041} C_VEL
LIN {X 0,Y 390.612,Z 303.788,A -85,B 0,C 180,E1 -11662.341,E2 -11662.341} C_VEL
LIN {X 0,Y 390.57,Z 303.528,A -85,B 0,C 180,E1 -11665.867,E2 -11665.867} C_VEL
LIN {X 0,Y 390.584,Z 303.939,A -85,B 0,C 180,E1 -11668.546,E2 -11668.546} C_VEL
LIN {X 0,Y 390.82,Z 305.041,A -85,B 0,C 180,E1 -11672.125,E2 -11672.125} C_VEL
LIN {X 0,Y 390.877,Z 306.076,A -85,B 0,C 180,E1 -11674.436,E2 -11674.436} C_VEL
LIN {X 0,Y 390.862,Z 307.277,A -85,B 0,C 180,E1 -11676.698,E2 -11676.698} C_VEL
LIN {X 0,Y 390.677,Z 309.326,A -85,B 0,C 180,E1 -11680.014,E2 -11680.014} C_VEL
LIN {X 0,Y 390.596,Z 310.094,A -85,B 0,C 180,E1 -11681.151,E2 -11681.151} C_VEL
LIN {X 0,Y 395.31,Z 322.571,A -85,B 0,C 180,E1 -11682.101,E2 -11682.101} C_VEL
LIN {X 0,Y 396.581,Z 327.257,A -85,B 0,C 180,E1 -11682.466,E2 -11682.466} C_VEL
LIN {X 0,Y 395.928,Z 338.887,A -85,B 0,C 180,E1 -11683.235,E2 -11683.235} C_VEL
LIN {X 0,Y 395.004,Z 351.205,A -85,B 0,C 180,E1 -11684.278,E2 -11684.278} C_VEL
LIN {X 0,Y 394.028,Z 362.891,A -85,B 0,C 180,E1 -11685.54,E2 -11685.54} C_VEL
LIN {X 0,Y 393.128,Z 372.395,A -85,B 0,C 180,E1 -11686.825,E2 -11686.825} C_VEL
LIN {X 0,Y 392.297,Z 381.671,A -85,B 0,C 180,E1 -11688.373,E2 -11688.373} C_VEL
LIN {X 0,Y 391.464,Z 389.045,A -85,B 0,C 180,E1 -11689.919,E2 -11689.919} C_VEL
LIN {X 0,Y 390.893,Z 394.814,A -85,B 0,C 180,E1 -11691.443,E2 -11691.443} C_VEL
LIN {X 0,Y 390.191,Z 400.194,A -85,B 0,C 180,E1 -11693.277,E2 -11693.277} C_VEL
LIN {X 0,Y 389.972,Z 403.463,A -85,B 0,C 180,E1 -11694.83,E2 -11694.83} C_VEL
LIN {X 0,Y 389.698,Z 405.064,A -85,B 0,C 180,E1 -11695.863,E2 -11695.863} C_VEL
LIN {X 0,Y 389.401,Z 406.242,A -85,B 0,C 180,E1 -11696.896,E2 -11696.896} C_VEL
LIN {X 0,Y 389.201,Z 407.005,A -85,B 0,C 180,E1 -11697.93,E2 -11697.93} C_VEL
LIN {X 0,Y 389.104,Z 407.318,A -85,B 0,C 180,E1 -11698.965,E2 -11698.965} C_VEL
LIN {X 0,Y 389.063,Z 407.197,A -85,B 0,C 180,E1 -11700,E2 -11700} C_VEL
LIN {X 0,Y 389.077,Z 406.672,A -85,B 0,C 180,E1 -11701.035,E2 -11701.035} C_VEL
LIN {X 0,Y 389.177,Z 405.73,A -85,B 0,C 180,E1 -11702.07,E2 -11702.07} C_VEL
LIN {X 0,Y 389.362,Z 404.319,A -85,B 0,C 180,E1 -11703.104,E2 -11703.104} C_VEL
LIN {X 0,Y 389.569,Z 401.413,A -85,B 0,C 180,E1 -11704.657,E2 -11704.657} C_VEL
LIN {X 0,Y 389.608,Z 397.456,A -85,B 0,C 180,E1 -11706.213,E2 -11706.213} C_VEL
LIN {X 0,Y 389.955,Z 392.31,A -85,B 0,C 180,E1 -11707.768,E2 -11707.768} C_VEL
LIN {X 0,Y 390.346,Z 385.845,A -85,B 0,C 180,E1 -11709.325,E2 -11709.325} C_VEL
LIN {X 0,Y 390.885,Z 377.815,A -85,B 0,C 180,E1 -11710.882,E2 -11710.882} C_VEL
LIN {X 0,Y 391.534,Z 367.778,A -85,B 0,C 180,E1 -11712.439,E2 -11712.439} C_VEL
LIN {X 0,Y 392.264,Z 357.43,A -85,B 0,C 180,E1 -11713.733,E2 -11713.733} C_VEL
LIN {X 0,Y 392.836,Z 346.235,A -85,B 0,C 180,E1 -11714.865,E2 -11714.865} C_VEL
LIN {X 0,Y 393.381,Z 334.628,A -85,B 0,C 180,E1 -11715.81,E2 -11715.81} C_VEL
LIN {X 0,Y 393.977,Z 322.286,A -85,B 0,C 180,E1 -11716.584,E2 -11716.584} C_VEL
LIN {X 0,Y 391.141,Z 309.506,A -85,B 0,C 180,E1 -11717.3,E2 -11717.3} C_VEL
LIN {X 0,Y 389.353,Z 301.896,A -85,B 0,C 180,E1 -11717.64,E2 -11717.64} C_VEL
LIN {X 0,Y 389.383,Z 300.985,A -85,B 0,C 180,E1 -11718.959,E2 -11718.959} C_VEL
LIN {X 0,Y 389.652,Z 300.944,A -85,B 0,C 180,E1 -11721.145,E2 -11721.145} C_VEL
LIN {X 0,Y 389.953,Z 300.913,A -85,B 0,C 180,E1 -11724.489,E2 -11724.489} C_VEL
LIN {X 0,Y 390.091,Z 300.888,A -85,B 0,C 180,E1 -11726.77,E2 -11726.77} C_VEL
LIN {X 0,Y 390.049,Z 300.899,A -85,B 0,C 180,E1 -11730.131,E2 -11730.131} C_VEL
LIN {X 0,Y 390.071,Z 300.898,A -85,B 0,C 180,E1 -11734.025,E2 -11734.025} C_VEL
LIN {X 0,Y 390.046,Z 300.9,A -85,B 0,C 180,E1 -11737.551,E2 -11737.551} C_VEL
LIN {X 0,Y 390.059,Z 300.899,A -85,B 0,C 180,E1 -11740.821,E2 -11740.821} C_VEL
LIN {X 0,Y 390.058,Z 300.901,A -85,B 0,C 180,E1 -11743.886,E2 -11743.886} C_VEL
LIN {X 0,Y 390.06,Z 300.894,A -85,B 0,C 180,E1 -11746.79,E2 -11746.79} C_VEL
LIN {X 0,Y 390.059,Z 300.9,A -85,B 0,C 180,E1 -11749.561,E2 -11749.561} C_VEL
LIN {X 0,Y 390.043,Z 300.899,A -85,B 0,C 180,E1 -11752.45,E2 -11752.45} C_VEL
LIN {X 0,Y 389.918,Z 300.921,A -85,B 0,C 180,E1 -11756.03,E2 -11756.03} C_VEL
LIN {X 0,Y 389.924,Z 300.966,A -85,B 0,C 180,E1 -11756.342,E2 -11756.342} C_VEL
LIN {X 0,Y 389.626,Z 306.743,A -85,B 0,C 180,E1 -11759.976,E2 -11759.976} C_VEL
LIN {X 0,Y 389.543,Z 311.829,A -85,B 0,C 180,E1 -11763.189,E2 -11763.189} C_VEL
LIN {X 0,Y 389.483,Z 317.983,A -85,B 0,C 180,E1 -11766.966,E2 -11766.966} C_VEL
LIN {X 0,Y 389.469,Z 323.131,A -85,B 0,C 180,E1 -11769.949,E2 -11769.949} C_VEL
LIN {X 0,Y 389.452,Z 326.012,A -85,B 0,C 180,E1 -11771.531,E2 -11771.531} C_VEL
LIN {X 0,Y 393.112,Z 340.032,A -85,B 0,C 180,E1 -11772.176,E2 -11772.176} C_VEL
LIN {X 0,Y 395.165,Z 350.042,A -85,B 0,C 180,E1 -11772.767,E2 -11772.767} C_VEL
LIN {X 0,Y 394.696,Z 360.953,A -85,B 0,C 180,E1 -11773.447,E2 -11773.447} C_VEL
LIN {X 0,Y 393.958,Z 372.188,A -85,B 0,C 180,E1 -11774.346,E2 -11774.346} C_VEL
LIN {X 0,Y 393.132,Z 383.499,A -85,B 0,C 180,E1 -11775.506,E2 -11775.506} C_VEL
LIN {X 0,Y 392.234,Z 393.582,A -85,B 0,C 180,E1 -11776.794,E2 -11776.794} C_VEL
LIN {X 0,Y 391.355,Z 403.199,A -85,B 0,C 180,E1 -11778.344,E2 -11778.344} C_VEL
LIN {X 0,Y 390.603,Z 410.929,A -85,B 0,C 180,E1 -11779.896,E2 -11779.896} C_VEL
LIN {X 0,Y 390.087,Z 416.148,A -85,B 0,C 180,E1 -11781.191,E2 -11781.191} C_VEL
LIN {X 0,Y 389.616,Z 421.4,A -85,B 0,C 180,E1 -11782.798,E2 -11782.798} C_VEL
LIN {X 0,Y 389.25,Z 425.195,A -85,B 0,C 180,E1 -11784.301,E2 -11784.301} C_VEL
LIN {X 0,Y 389.171,Z 428.096,A -85,B 0,C 180,E1 -11785.858,E2 -11785.858} C_VEL
LIN {X 0,Y 389.073,Z 429.506,A -85,B 0,C 180,E1 -11786.894,E2 -11786.894} C_VEL
LIN {X 0,Y 388.834,Z 431.114,A -85,B 0,C 180,E1 -11788.964,E2 -11788.964} C_VEL
LIN {X 0,Y 388.82,Z 431.348,A -85,B 0,C 180,E1 -11790,E2 -11790} C_VEL
LIN {X 0,Y 388.928,Z 430.573,A -85,B 0,C 180,E1 -11792.071,E2 -11792.071} C_VEL
LIN {X 0,Y 389.072,Z 429.607,A -85,B 0,C 180,E1 -11793.106,E2 -11793.106} C_VEL
LIN {X 0,Y 389.143,Z 428.255,A -85,B 0,C 180,E1 -11794.143,E2 -11794.143} C_VEL
LIN {X 0,Y 389.235,Z 425.41,A -85,B 0,C 180,E1 -11795.699,E2 -11795.699} C_VEL
LIN {X 0,Y 389.619,Z 421.532,A -85,B 0,C 180,E1 -11797.254,E2 -11797.254} C_VEL
LIN {X 0,Y 390.041,Z 416.513,A -85,B 0,C 180,E1 -11798.81,E2 -11798.81} C_VEL
LIN {X 0,Y 390.685,Z 410.172,A -85,B 0,C 180,E1 -11800.363,E2 -11800.363} C_VEL
LIN {X 0,Y 391.413,Z 402.293,A -85,B 0,C 180,E1 -11801.917,E2 -11801.917} C_VEL
LIN {X 0,Y 392.187,Z 394.237,A -85,B 0,C 180,E1 -11803.208,E2 -11803.208} C_VEL
LIN {X 0,Y 393.1,Z 384.346,A -85,B 0,C 180,E1 -11804.495,E2 -11804.495} C_VEL
LIN {X 0,Y 393.861,Z 373.207,A -85,B 0,C 180,E1 -11805.658,E2 -11805.658} C_VEL
LIN {X 0,Y 393.905,Z 372.587,A -85,B 0,C 180,E1 -11805.716,E2 -11805.716} C_VEL
LIN {X 0,Y 393.697,Z 367.608,A -85,B 0,C 180,E1 -11806.182,E2 -11806.182} C_VEL
LIN {X 0,Y 391.617,Z 359.375,A -85,B 0,C 180,E1 -11806.928,E2 -11806.928} C_VEL
LIN {X 0,Y 389.31,Z 352.656,A -85,B 0,C 180,E1 -11807.477,E2 -11807.477} C_VEL
LIN {X 0,Y 387.317,Z 345.608,A -85,B 0,C 180,E1 -11807.956,E2 -11807.956} C_VEL
LIN {X 0,Y 384.14,Z 332.576,A -85,B 0,C 180,E1 -11808.652,E2 -11808.652} C_VEL
LIN {X 0,Y 382.426,Z 326.371,A -85,B 0,C 180,E1 -11808.934,E2 -11808.934} C_VEL
LIN {X 0,Y 382.421,Z 321.666,A -85,B 0,C 180,E1 -11811.565,E2 -11811.565} C_VEL
LIN {X 0,Y 382.451,Z 315.922,A -85,B 0,C 180,E1 -11815.002,E2 -11815.002} C_VEL
LIN {X 0,Y 382.555,Z 310.278,A -85,B 0,C 180,E1 -11818.532,E2 -11818.532} C_VEL
LIN {X 0,Y 382.721,Z 304.537,A -85,B 0,C 180,E1 -11822.177,E2 -11822.177} C_VEL
LIN {X 0,Y 382.904,Z 301.793,A -85,B 0,C 180,E1 -11824.01,E2 -11824.01} C_VEL
LIN {X 0,Y 382.99,Z 301.781,A -85,B 0,C 180,E1 -11827.269,E2 -11827.269} C_VEL
LIN {X 0,Y 383.011,Z 301.778,A -85,B 0,C 180,E1 -11829.958,E2 -11829.958} C_VEL
LIN {X 0,Y 383.007,Z 301.78,A -85,B 0,C 180,E1 -11832.779,E2 -11832.779} C_VEL
LIN {X 0,Y 383,Z 301.779,A -85,B 0,C 180,E1 -11835.789,E2 -11835.789} C_VEL
LIN {X 0,Y 382.991,Z 301.777,A -85,B 0,C 180,E1 -11838.796,E2 -11838.796} C_VEL
LIN {X 0,Y 382.999,Z 301.775,A -85,B 0,C 180,E1 -11842.097,E2 -11842.097} C_VEL
LIN {X 0,Y 382.958,Z 301.784,A -85,B 0,C 180,E1 -11844.037,E2 -11844.037} C_VEL
LIN {X 0,Y 382.716,Z 301.93,A -85,B 0,C 180,E1 -11847.1,E2 -11847.1} C_VEL
LIN {X 0,Y 382.461,Z 307.038,A -85,B 0,C 180,E1 -11850.255,E2 -11850.255} C_VEL
LIN {X 0,Y 382.383,Z 310.905,A -85,B 0,C 180,E1 -11852.646,E2 -11852.646} C_VEL
LIN {X 0,Y 382.332,Z 314.7,A -85,B 0,C 180,E1 -11854.989,E2 -11854.989} C_VEL
LIN {X 0,Y 382.285,Z 320.305,A -85,B 0,C 180,E1 -11858.427,E2 -11858.427} C_VEL
LIN {X 0,Y 382.196,Z 326.512,A -85,B 0,C 180,E1 -11862.217,E2 -11862.217} C_VEL
LIN {X 0,Y 384.948,Z 339.803,A -85,B 0,C 180,E1 -11862.834,E2 -11862.834} C_VEL
LIN {X 0,Y 386.658,Z 348.816,A -85,B 0,C 180,E1 -11863.365,E2 -11863.365} C_VEL
LIN {X 0,Y 386.041,Z 360.885,A -85,B 0,C 180,E1 -11864.152,E2 -11864.152} C_VEL
LIN {X 0,Y 385.348,Z 373.463,A -85,B 0,C 180,E1 -11865.207,E2 -11865.207} C_VEL
LIN {X 0,Y 384.741,Z 384.622,A -85,B 0,C 180,E1 -11866.397,E2 -11866.397} C_VEL
LIN {X 0,Y 384.049,Z 393.793,A -85,B 0,C 180,E1 -11867.583,E2 -11867.583} C_VEL
LIN {X 0,Y 383.501,Z 402.244,A -85,B 0,C 180,E1 -11868.906,E2 -11868.906} C_VEL
LIN {X 0,Y 382.925,Z 410.486,A -85,B 0,C 180,E1 -11870.492,E2 -11870.492} C_VEL
LIN {X 0,Y 382.499,Z 417.152,A -85,B 0,C 180,E1 -11872.079,E2 -11872.079} C_VEL
LIN {X 0,Y 382.213,Z 422.42,A -85,B 0,C 180,E1 -11873.666,E2 -11873.666} C_VEL
LIN {X 0,Y 382.01,Z 426.474,A -85,B 0,C 180,E1 -11875.251,E2 -11875.251} C_VEL
LIN {X 0,Y 381.989,Z 429.443,A -85,B 0,C 180,E1 -11876.836,E2 -11876.836} C_VEL
LIN {X 0,Y 381.864,Z 430.861,A -85,B 0,C 180,E1 -11877.89,E2 -11877.89} C_VEL
LIN {X 0,Y 381.784,Z 431.872,A -85,B 0,C 180,E1 -11878.945,E2 -11878.945} C_VEL
LIN {X 0,Y 381.782,Z 432.405,A -85,B 0,C 180,E1 -11880,E2 -11880} C_VEL
LIN {X 0,Y 381.824,Z 432.526,A -85,B 0,C 180,E1 -11881.055,E2 -11881.055} C_VEL
LIN {X 0,Y 381.931,Z 432.238,A -85,B 0,C 180,E1 -11882.109,E2 -11882.109} C_VEL
LIN {X 0,Y 382.069,Z 431.478,A -85,B 0,C 180,E1 -11883.163,E2 -11883.163} C_VEL
LIN {X 0,Y 382.245,Z 430.298,A -85,B 0,C 180,E1 -11884.218,E2 -11884.218} C_VEL
LIN {X 0,Y 382.35,Z 427.716,A -85,B 0,C 180,E1 -11885.802,E2 -11885.802} C_VEL
LIN {X 0,Y 382.838,Z 423.606,A -85,B 0,C 180,E1 -11887.556,E2 -11887.556} C_VEL
LIN {X 0,Y 383.348,Z 419.235,A -85,B 0,C 180,E1 -11888.965,E2 -11888.965} C_VEL
LIN {X 0,Y 383.981,Z 413.062,A -85,B 0,C 180,E1 -11890.546,E2 -11890.546} C_VEL
LIN {X 0,Y 384.715,Z 405.34,A -85,B 0,C 180,E1 -11892.127,E2 -11892.127} C_VEL
LIN {X 0,Y 385.53,Z 397.511,A -85,B 0,C 180,E1 -11893.44,E2 -11893.44} C_VEL
LIN {X 0,Y 386.463,Z 387.951,A -85,B 0,C 180,E1 -11894.75,E2 -11894.75} C_VEL
LIN {X 0,Y 387.5,Z 376.665,A -85,B 0,C 180,E1 -11896.002,E2 -11896.002} C_VEL
LIN {X 0,Y 388.502,Z 364.12,A -85,B 0,C 180,E1 -11897.095,E2 -11897.095} C_VEL
LIN {X 0,Y 389.304,Z 352.864,A -85,B 0,C 180,E1 -11897.872,E2 -11897.872} C_VEL
LIN {X 0,Y 387.656,Z 344.932,A -85,B 0,C 180,E1 -11898.463,E2 -11898.463} C_VEL
LIN {X 0,Y 383.864,Z 333.246,A -85,B 0,C 180,E1 -11899.303,E2 -11899.303} C_VEL
LIN {X 0,Y 383.126,Z 330.857,A -85,B 0,C 180,E1 -11899.454,E2 -11899.454} C_VEL
LIN {X 0,Y 383.288,Z 324.059,A -85,B 0,C 180,E1 -11903.536,E2 -11903.536} C_VEL
LIN {X 0,Y 383.456,Z 317.768,A -85,B 0,C 180,E1 -11907.271,E2 -11907.271} C_VEL
LIN {X 0,Y 383.726,Z 311.904,A -85,B 0,C 180,E1 -11910.592,E2 -11910.592} C_VEL
LIN {X 0,Y 383.906,Z 307.084,A -85,B 0,C 180,E1 -11913.312,E2 -11913.312} C_VEL
LIN {X 0,Y 383.011,Z 301.778,A -85,B 0,C 180,E1 -11916.436,E2 -11916.436} C_VEL
LIN {X 0,Y 383.009,Z 301.777,A -85,B 0,C 180,E1 -11919.958,E2 -11919.958} C_VEL
LIN {X 0,Y 383.04,Z 301.773,A -85,B 0,C 180,E1 -11924.067,E2 -11924.067} C_VEL
LIN {X 0,Y 384.545,Z 309.779,A -85,B 0,C 180,E1 -11927.89,E2 -11927.89} C_VEL
LIN {X 0,Y 386.124,Z 317.768,A -85,B 0,C 180,E1 -11931.505,E2 -11931.505} C_VEL
LIN {X 0,Y 386.573,Z 321.55,A -85,B 0,C 180,E1 -11933.134,E2 -11933.134} C_VEL
LIN {X 0,Y 386.034,Z 327.749,A -85,B 0,C 180,E1 -11935.641,E2 -11935.641} C_VEL
LIN {X 0,Y 385.156,Z 337.008,A -85,B 0,C 180,E1 -11939.275,E2 -11939.275} C_VEL
LIN {X 0,Y 384.201,Z 347.57,A -85,B 0,C 180,E1 -11943.305,E2 -11943.305} C_VEL
LIN {X 0,Y 383.621,Z 355.742,A -85,B 0,C 180,E1 -11946.35,E2 -11946.35} C_VEL
LIN {X 0,Y 382.948,Z 366.067,A -85,B 0,C 180,E1 -11950.152,E2 -11950.152} C_VEL
LIN {X 0,Y 382.803,Z 368.625,A -85,B 0,C 180,E1 -11951.086,E2 -11951.086} C_VEL
LIN {X 0,Y 384.913,Z 382.983,A -85,B 0,C 180,E1 -11951.705,E2 -11951.705} C_VEL
LIN {X 0,Y 386.295,Z 394.716,A -85,B 0,C 180,E1 -11952.376,E2 -11952.376} C_VEL
LIN {X 0,Y 387.1,Z 401.91,A -85,B 0,C 180,E1 -11952.88,E2 -11952.88} C_VEL
LIN {X 0,Y 386.262,Z 413.219,A -85,B 0,C 180,E1 -11953.755,E2 -11953.755} C_VEL
LIN {X 0,Y 385.318,Z 424.028,A -85,B 0,C 180,E1 -11954.8,E2 -11954.8} C_VEL
LIN {X 0,Y 384.47,Z 434.614,A -85,B 0,C 180,E1 -11956.081,E2 -11956.081} C_VEL
LIN {X 0,Y 383.583,Z 444.552,A -85,B 0,C 180,E1 -11957.568,E2 -11957.568} C_VEL
LIN {X 0,Y 382.803,Z 453.047,A -85,B 0,C 180,E1 -11959.153,E2 -11959.153} C_VEL
LIN {X 0,Y 382.323,Z 459.898,A -85,B 0,C 180,E1 -11960.744,E2 -11960.744} C_VEL
LIN {X 0,Y 381.959,Z 466.173,A -85,B 0,C 180,E1 -11962.6,E2 -11962.6} C_VEL
LIN {X 0,Y 381.828,Z 469.873,A -85,B 0,C 180,E1 -11964.021,E2 -11964.021} C_VEL
LIN {X 0,Y 381.693,Z 473.282,A -85,B 0,C 180,E1 -11965.776,E2 -11965.776} C_VEL
LIN {X 0,Y 381.761,Z 474.785,A -85,B 0,C 180,E1 -11966.834,E2 -11966.834} C_VEL
LIN {X 0,Y 381.774,Z 475.862,A -85,B 0,C 180,E1 -11967.89,E2 -11967.89} C_VEL
LIN {X 0,Y 381.83,Z 476.544,A -85,B 0,C 180,E1 -11968.945,E2 -11968.945} C_VEL
LIN {X 0,Y 381.824,Z 476.778,A -85,B 0,C 180,E1 -11970,E2 -11970} C_VEL
LIN {X 0,Y 381.821,Z 476.558,A -85,B 0,C 180,E1 -11971.055,E2 -11971.055} C_VEL
LIN {X 0,Y 381.789,Z 475.929,A -85,B 0,C 180,E1 -11972.11,E2 -11972.11} C_VEL
LIN {X 0,Y 381.739,Z 474.874,A -85,B 0,C 180,E1 -11973.166,E2 -11973.166} C_VEL
LIN {X 0,Y 381.709,Z 473.335,A -85,B 0,C 180,E1 -11974.224,E2 -11974.224} C_VEL
LIN {X 0,Y 381.829,Z 469.771,A -85,B 0,C 180,E1 -11975.992,E2 -11975.992} C_VEL
LIN {X 0,Y 382.032,Z 464.408,A -85,B 0,C 180,E1 -11977.931,E2 -11977.931} C_VEL
LIN {X 0,Y 382.418,Z 458.72,A -85,B 0,C 180,E1 -11979.521,E2 -11979.521} C_VEL
LIN {X 0,Y 382.92,Z 451.556,A -85,B 0,C 180,E1 -11981.111,E2 -11981.111} C_VEL
LIN {X 0,Y 383.734,Z 442.615,A -85,B 0,C 180,E1 -11982.696,E2 -11982.696} C_VEL
LIN {X 0,Y 384.557,Z 433.033,A -85,B 0,C 180,E1 -11984.068,E2 -11984.068} C_VEL
LIN {X 0,Y 385.362,Z 422.659,A -85,B 0,C 180,E1 -11985.334,E2 -11985.334} C_VEL
LIN {X 0,Y 386.515,Z 410.676,A -85,B 0,C 180,E1 -11986.506,E2 -11986.506} C_VEL
LIN {X 0,Y 387.158,Z 400.886,A -85,B 0,C 180,E1 -11987.293,E2 -11987.293} C_VEL
LIN {X 0,Y 386.03,Z 389.132,A -85,B 0,C 180,E1 -11988.153,E2 -11988.153} C_VEL
LIN {X 0,Y 384.7,Z 375.421,A -85,B 0,C 180,E1 -11988.952,E2 -11988.952} C_VEL
LIN {X 0,Y 382.735,Z 364.428,A -85,B 0,C 180,E1 -11989.51,E2 -11989.51} C_VEL
LIN {X 0,Y 383.299,Z 354.485,A -85,B 0,C 180,E1 -11993.104,E2 -11993.104} C_VEL
LIN {X 0,Y 383.822,Z 346.24,A -85,B 0,C 180,E1 -11996.205,E2 -11996.205} C_VEL
LIN {X 0,Y 384.544,Z 337.723,A -85,B 0,C 180,E1 -11999.568,E2 -11999.568} C_VEL
LIN {X 0,Y 385.282,Z 330.828,A -85,B 0,C 180,E1 -12002.47,E2 -12002.47} C_VEL
LIN {X 0,Y 386.273,Z 323.969,A -85,B 0,C 180,E1 -12005.607,E2 -12005.607} C_VEL
LIN {X 0,Y 386.49,Z 320.231,A -85,B 0,C 180,E1 -12007.53,E2 -12007.53} C_VEL
LIN {X 0,Y 385.806,Z 316.051,A -85,B 0,C 180,E1 -12010.085,E2 -12010.085} C_VEL
LIN {X 0,Y 385.012,Z 312.005,A -85,B 0,C 180,E1 -12013.1,E2 -12013.1} C_VEL
LIN {X 0,Y 384.445,Z 309.052,A -85,B 0,C 180,E1 -12015.999,E2 -12015.999} C_VEL
LIN {X 0,Y 384.066,Z 307.045,A -85,B 0,C 180,E1 -12018.794,E2 -12018.794} C_VEL
LIN {X 0,Y 383.782,Z 305.726,A -85,B 0,C 180,E1 -12021.947,E2 -12021.947} C_VEL
LIN {X 0,Y 383.677,Z 305.277,A -85,B 0,C 180,E1 -12025.4,E2 -12025.4} C_VEL
LIN {X 0,Y 383.683,Z 305.5,A -85,B 0,C 180,E1 -12027.913,E2 -12027.913} C_VEL
LIN {X 0,Y 383.821,Z 306.429,A -85,B 0,C 180,E1 -12031.571,E2 -12031.571} C_VEL
LIN {X 0,Y 383.934,Z 307.37,A -85,B 0,C 180,E1 -12033.939,E2 -12033.939} C_VEL
LIN {X 0,Y 383.874,Z 309.135,A -85,B 0,C 180,E1 -12037.389,E2 -12037.389} C_VEL
LIN {X 0,Y 383.675,Z 311.253,A -85,B 0,C 180,E1 -12040.662,E2 -12040.662} C_VEL
LIN {X 0,Y 388.772,Z 324.378,A -85,B 0,C 180,E1 -12041.725,E2 -12041.725} C_VEL
LIN {X 0,Y 390.059,Z 328.522,A -85,B 0,C 180,E1 -12042.075,E2 -12042.075} C_VEL
LIN {X 0,Y 389.314,Z 341.344,A -85,B 0,C 180,E1 -12042.969,E2 -12042.969} C_VEL
LIN {X 0,Y 388.24,Z 354.133,A -85,B 0,C 180,E1 -12044.121,E2 -12044.121} C_VEL
LIN {X 0,Y 387.327,Z 364.413,A -85,B 0,C 180,E1 -12045.284,E2 -12045.284} C_VEL
LIN {X 0,Y 386.362,Z 373.788,A -85,B 0,C 180,E1 -12046.59,E2 -12046.59} C_VEL
LIN {X 0,Y 385.454,Z 382.89,A -85,B 0,C 180,E1 -12048.163,E2 -12048.163} C_VEL
LIN {X 0,Y 384.584,Z 390.159,A -85,B 0,C 180,E1 -12049.737,E2 -12049.737} C_VEL
LIN {X 0,Y 383.969,Z 395.793,A -85,B 0,C 180,E1 -12051.263,E2 -12051.263} C_VEL
LIN {X 0,Y 383.359,Z 399.836,A -85,B 0,C 180,E1 -12052.627,E2 -12052.627} C_VEL
LIN {X 0,Y 383.015,Z 403.394,A -85,B 0,C 180,E1 -12054.208,E2 -12054.208} C_VEL
LIN {X 0,Y 382.676,Z 405.911,A -85,B 0,C 180,E1 -12055.787,E2 -12055.787} C_VEL
LIN {X 0,Y 382.368,Z 407.059,A -85,B 0,C 180,E1 -12056.839,E2 -12056.839} C_VEL
LIN {X 0,Y 382.155,Z 407.79,A -85,B 0,C 180,E1 -12057.892,E2 -12057.892} C_VEL
LIN {X 0,Y 382.05,Z 408.052,A -85,B 0,C 180,E1 -12058.946,E2 -12058.946} C_VEL
LIN {X 0,Y 382.007,Z 407.896,A -85,B 0,C 180,E1 -12060,E2 -12060} C_VEL
LIN {X 0,Y 382.024,Z 407.333,A -85,B 0,C 180,E1 -12061.054,E2 -12061.054} C_VEL
LIN {X 0,Y 382.132,Z 406.332,A -85,B 0,C 180,E1 -12062.108,E2 -12062.108} C_VEL
LIN {X 0,Y 382.293,Z 404.882,A -85,B 0,C 180,E1 -12063.162,E2 -12063.162} C_VEL
LIN {X 0,Y 382.523,Z 401.901,A -85,B 0,C 180,E1 -12064.743,E2 -12064.743} C_VEL
LIN {X 0,Y 382.57,Z 397.867,A -85,B 0,C 180,E1 -12066.328,E2 -12066.328} C_VEL
LIN {X 0,Y 382.994,Z 391.673,A -85,B 0,C 180,E1 -12068.176,E2 -12068.176} C_VEL
LIN {X 0,Y 383.423,Z 384.85,A -85,B 0,C 180,E1 -12069.762,E2 -12069.762} C_VEL
LIN {X 0,Y 384.016,Z 376.387,A -85,B 0,C 180,E1 -12071.346,E2 -12071.346} C_VEL
LIN {X 0,Y 384.581,Z 367.776,A -85,B 0,C 180,E1 -12072.668,E2 -12072.668} C_VEL
LIN {X 0,Y 385.313,Z 357.227,A -85,B 0,C 180,E1 -12073.986,E2 -12073.986} C_VEL
LIN {X 0,Y 385.96,Z 345.361,A -85,B 0,C 180,E1 -12075.184,E2 -12075.184} C_VEL
LIN {X 0,Y 386.515,Z 333.958,A -85,B 0,C 180,E1 -12076.099,E2 -12076.099} C_VEL
LIN {X 0,Y 386.957,Z 322.44,A -85,B 0,C 180,E1 -12076.826,E2 -12076.826} C_VEL
LIN {X 0,Y 383.815,Z 308.907,A -85,B 0,C 180,E1 -12077.597,E2 -12077.597} C_VEL
LIN {X 0,Y 382.308,Z 302.464,A -85,B 0,C 180,E1 -12077.891,E2 -12077.891} C_VEL
LIN {X 0,Y 382.297,Z 301.868,A -85,B 0,C 180,E1 -12078.489,E2 -12078.489} C_VEL
LIN {X 0,Y 382.635,Z 301.818,A -85,B 0,C 180,E1 -12081.552,E2 -12081.552} C_VEL
LIN {X 0,Y 382.935,Z 301.783,A -85,B 0,C 180,E1 -12084.969,E2 -12084.969} C_VEL
LIN {X 0,Y 383.027,Z 301.772,A -85,B 0,C 180,E1 -12088.269,E2 -12088.269} C_VEL
LIN {X 0,Y 383.012,Z 301.772,A -85,B 0,C 180,E1 -12092.15,E2 -12092.15} C_VEL
LIN {X 0,Y 383.021,Z 301.77,A -85,B 0,C 180,E1 -12094.668,E2 -12094.668} C_VEL
LIN {X 0,Y 383.002,Z 301.781,A -85,B 0,C 180,E1 -12097.904,E2 -12097.904} C_VEL
LIN {X 0,Y 382.986,Z 301.78,A -85,B 0,C 180,E1 -12101.347,E2 -12101.347} C_VEL
LIN {X 0,Y 382.999,Z 301.777,A -85,B 0,C 180,E1 -12104.304,E2 -12104.304} C_VEL
LIN {X 0,Y 383.012,Z 301.773,A -85,B 0,C 180,E1 -12107.24,E2 -12107.24} C_VEL
LIN {X 0,Y 383.017,Z 301.775,A -85,B 0,C 180,E1 -12110.414,E2 -12110.414} C_VEL
LIN {X 0,Y 382.971,Z 301.784,A -85,B 0,C 180,E1 -12114.038,E2 -12114.038} C_VEL
LIN {X 0,Y 382.898,Z 301.921,A -85,B 0,C 180,E1 -12116.29,E2 -12116.29} C_VEL
LIN {X 0,Y 382.571,Z 308.194,A -85,B 0,C 180,E1 -12120.264,E2 -12120.264} C_VEL
LIN {X 0,Y 382.517,Z 311.969,A -85,B 0,C 180,E1 -12122.656,E2 -12122.656} C_VEL
LIN {X 0,Y 382.436,Z 317.634,A -85,B 0,C 180,E1 -12126.153,E2 -12126.153} C_VEL
LIN {X 0,Y 382.408,Z 323.524,A -85,B 0,C 180,E1 -12129.602,E2 -12129.602} C_VEL
LIN {X 0,Y 382.414,Z 326.356,A -85,B 0,C 180,E1 -12131.17,E2 -12131.17} C_VEL
LIN {X 0,Y 386.265,Z 341.126,A -85,B 0,C 180,E1 -12131.878,E2 -12131.878} C_VEL
LIN {X 0,Y 388.399,Z 351.202,A -85,B 0,C 180,E1 -12132.5,E2 -12132.5} C_VEL
LIN {X 0,Y 387.768,Z 363.132,A -85,B 0,C 180,E1 -12133.278,E2 -12133.278} C_VEL
LIN {X 0,Y 386.897,Z 375.233,A -85,B 0,C 180,E1 -12134.313,E2 -12134.313} C_VEL
LIN {X 0,Y 386.096,Z 386.121,A -85,B 0,C 180,E1 -12135.505,E2 -12135.505} C_VEL
LIN {X 0,Y 385.164,Z 395.728,A -85,B 0,C 180,E1 -12136.816,E2 -12136.816} C_VEL
LIN {X 0,Y 384.243,Z 405.05,A -85,B 0,C 180,E1 -12138.393,E2 -12138.393} C_VEL
LIN {X 0,Y 383.49,Z 412.447,A -85,B 0,C 180,E1 -12139.974,E2 -12139.974} C_VEL
LIN {X 0,Y 382.913,Z 418.384,A -85,B 0,C 180,E1 -12141.557,E2 -12141.557} C_VEL
LIN {X 0,Y 382.511,Z 423.087,A -85,B 0,C 180,E1 -12143.146,E2 -12143.146} C_VEL
LIN {X 0,Y 382.102,Z 426.671,A -85,B 0,C 180,E1 -12144.723,E2 -12144.723} C_VEL
LIN {X 0,Y 382.087,Z 428.512,A -85,B 0,C 180,E1 -12145.781,E2 -12145.781} C_VEL
LIN {X 0,Y 382.017,Z 429.92,A -85,B 0,C 180,E1 -12146.836,E2 -12146.836} C_VEL
LIN {X 0,Y 381.763,Z 431.528,A -85,B 0,C 180,E1 -12148.945,E2 -12148.945} C_VEL
LIN {X 0,Y 381.746,Z 431.762,A -85,B 0,C 180,E1 -12150,E2 -12150} C_VEL
LIN {X 0,Y 381.864,Z 430.986,A -85,B 0,C 180,E1 -12152.109,E2 -12152.109} C_VEL
LIN {X 0,Y 382.014,Z 430.02,A -85,B 0,C 180,E1 -12153.164,E2 -12153.164} C_VEL
LIN {X 0,Y 382.06,Z 428.669,A -85,B 0,C 180,E1 -12154.22,E2 -12154.22} C_VEL
LIN {X 0,Y 382.201,Z 425.822,A -85,B 0,C 180,E1 -12155.805,E2 -12155.805} C_VEL
LIN {X 0,Y 382.596,Z 421.944,A -85,B 0,C 180,E1 -12157.388,E2 -12157.388} C_VEL
LIN {X 0,Y 383.028,Z 416.925,A -85,B 0,C 180,E1 -12158.973,E2 -12158.973} C_VEL
LIN {X 0,Y 383.719,Z 410.581,A -85,B 0,C 180,E1 -12160.554,E2 -12160.554} C_VEL
LIN {X 0,Y 384.492,Z 402.699,A -85,B 0,C 180,E1 -12162.134,E2 -12162.134} C_VEL
LIN {X 0,Y 385.309,Z 394.641,A -85,B 0,C 180,E1 -12163.448,E2 -12163.448} C_VEL
LIN {X 0,Y 386.257,Z 384.745,A -85,B 0,C 180,E1 -12164.758,E2 -12164.758} C_VEL
LIN {X 0,Y 386.929,Z 374.977,A -85,B 0,C 180,E1 -12165.81,E2 -12165.81} C_VEL
LIN {X 0,Y 387.718,Z 364.373,A -85,B 0,C 180,E1 -12166.724,E2 -12166.724} C_VEL
LIN {X 0,Y 388.383,Z 353.436,A -85,B 0,C 180,E1 -12167.464,E2 -12167.464} C_VEL
LIN {X 0,Y 388.197,Z 349.842,A -85,B 0,C 180,E1 -12167.685,E2 -12167.685} C_VEL
LIN {X 0,Y 387.317,Z 345.608,A -85,B 0,C 180,E1 -12167.956,E2 -12167.956} C_VEL
LIN {X 0,Y 385.846,Z 342.248,A -85,B 0,C 180,E1 -12168.192,E2 -12168.192} C_VEL
LIN {X 0,Y 377.575,Z 332.913,A -85,B 0,C 180,E1 -12168.994,E2 -12168.994} C_VEL
LIN {X 0,Y 376.097,Z 329.422,A -85,B 0,C 180,E1 -12169.174,E2 -12169.174} C_VEL
LIN {X 0,Y 375.4,Z 326.706,A -85,B 0,C 180,E1 -12169.312,E2 -12169.312} C_VEL
LIN {X 0,Y 375.394,Z 321.97,A -85,B 0,C 180,E1 -12171.989,E2 -12171.989} C_VEL
LIN {X 0,Y 375.431,Z 316.132,A -85,B 0,C 180,E1 -12175.503,E2 -12175.503} C_VEL
LIN {X 0,Y 375.534,Z 310.394,A -85,B 0,C 180,E1 -12179.116,E2 -12179.116} C_VEL
LIN {X 0,Y 375.742,Z 304.53,A -85,B 0,C 180,E1 -12182.849,E2 -12182.849} C_VEL
LIN {X 0,Y 375.859,Z 302.67,A -85,B 0,C 180,E1 -12184.122,E2 -12184.122} C_VEL
LIN {X 0,Y 375.937,Z 302.659,A -85,B 0,C 180,E1 -12186.743,E2 -12186.743} C_VEL
LIN {X 0,Y 375.991,Z 302.652,A -85,B 0,C 180,E1 -12189.971,E2 -12189.971} C_VEL
LIN {X 0,Y 375.932,Z 302.66,A -85,B 0,C 180,E1 -12193.766,E2 -12193.766} C_VEL
LIN {X 0,Y 375.936,Z 302.658,A -85,B 0,C 180,E1 -12196.811,E2 -12196.811} C_VEL
LIN {X 0,Y 375.965,Z 302.654,A -85,B 0,C 180,E1 -12200.538,E2 -12200.538} C_VEL
LIN {X 0,Y 375.915,Z 302.66,A -85,B 0,C 180,E1 -12203.506,E2 -12203.506} C_VEL
LIN {X 0,Y 375.684,Z 302.691,A -85,B 0,C 180,E1 -12206.986,E2 -12206.986} C_VEL
LIN {X 0,Y 375.389,Z 308.893,A -85,B 0,C 180,E1 -12210.871,E2 -12210.871} C_VEL
LIN {X 0,Y 375.302,Z 314.696,A -85,B 0,C 180,E1 -12214.488,E2 -12214.488} C_VEL
LIN {X 0,Y 375.242,Z 320.314,A -85,B 0,C 180,E1 -12218.001,E2 -12218.001} C_VEL
LIN {X 0,Y 375.174,Z 326.684,A -85,B 0,C 180,E1 -12221.854,E2 -12221.854} C_VEL
LIN {X 0,Y 375.175,Z 326.856,A -85,B 0,C 180,E1 -12221.96,E2 -12221.96} C_VEL
LIN {X 0,Y 378.222,Z 341.922,A -85,B 0,C 180,E1 -12222.704,E2 -12222.704} C_VEL
LIN {X 0,Y 379.725,Z 349.888,A -85,B 0,C 180,E1 -12223.19,E2 -12223.19} C_VEL
LIN {X 0,Y 379.006,Z 363.513,A -85,B 0,C 180,E1 -12224.126,E2 -12224.126} C_VEL
LIN {X 0,Y 378.287,Z 375.57,A -85,B 0,C 180,E1 -12225.203,E2 -12225.203} C_VEL
LIN {X 0,Y 377.651,Z 386.413,A -85,B 0,C 180,E1 -12226.411,E2 -12226.411} C_VEL
LIN {X 0,Y 376.94,Z 395.337,A -85,B 0,C 180,E1 -12227.619,E2 -12227.619} C_VEL
LIN {X 0,Y 376.286,Z 405.038,A -85,B 0,C 180,E1 -12229.235,E2 -12229.235} C_VEL
LIN {X 0,Y 375.73,Z 412.848,A -85,B 0,C 180,E1 -12230.852,E2 -12230.852} C_VEL
LIN {X 0,Y 375.263,Z 420.164,A -85,B 0,C 180,E1 -12232.775,E2 -12232.775} C_VEL
LIN {X 0,Y 375,Z 425.434,A -85,B 0,C 180,E1 -12234.623,E2 -12234.623} C_VEL
LIN {X 0,Y 374.918,Z 427.838,A -85,B 0,C 180,E1 -12235.7,E2 -12235.7} C_VEL
LIN {X 0,Y 374.913,Z 429.758,A -85,B 0,C 180,E1 -12236.776,E2 -12236.776} C_VEL
LIN {X 0,Y 374.801,Z 431.213,A -85,B 0,C 180,E1 -12237.851,E2 -12237.851} C_VEL
LIN {X 0,Y 374.714,Z 432.263,A -85,B 0,C 180,E1 -12238.925,E2 -12238.925} C_VEL
LIN {X 0,Y 374.708,Z 432.852,A -85,B 0,C 180,E1 -12240,E2 -12240} C_VEL
LIN {X 0,Y 374.752,Z 433.004,A -85,B 0,C 180,E1 -12241.075,E2 -12241.075} C_VEL
LIN {X 0,Y 374.865,Z 432.75,A -85,B 0,C 180,E1 -12242.149,E2 -12242.149} C_VEL
LIN {X 0,Y 375.016,Z 432.046,A -85,B 0,C 180,E1 -12243.223,E2 -12243.223} C_VEL
LIN {X 0,Y 375.207,Z 430.901,A -85,B 0,C 180,E1 -12244.297,E2 -12244.297} C_VEL
LIN {X 0,Y 375.323,Z 428.387,A -85,B 0,C 180,E1 -12245.911,E2 -12245.911} C_VEL
LIN {X 0,Y 375.825,Z 424.477,A -85,B 0,C 180,E1 -12247.643,E2 -12247.643} C_VEL
LIN {X 0,Y 376.399,Z 420.011,A -85,B 0,C 180,E1 -12249.132,E2 -12249.132} C_VEL
LIN {X 0,Y 377.058,Z 413.957,A -85,B 0,C 180,E1 -12250.742,E2 -12250.742} C_VEL
LIN {X 0,Y 377.85,Z 406.365,A -85,B 0,C 180,E1 -12252.351,E2 -12252.351} C_VEL
LIN {X 0,Y 378.713,Z 398.613,A -85,B 0,C 180,E1 -12253.686,E2 -12253.686} C_VEL
LIN {X 0,Y 379.709,Z 389.194,A -85,B 0,C 180,E1 -12255.018,E2 -12255.018} C_VEL
LIN {X 0,Y 380.893,Z 377.426,A -85,B 0,C 180,E1 -12256.367,E2 -12256.367} C_VEL
LIN {X 0,Y 381.891,Z 365.997,A -85,B 0,C 180,E1 -12257.401,E2 -12257.401} C_VEL
LIN {X 0,Y 382.774,Z 353.764,A -85,B 0,C 180,E1 -12258.28,E2 -12258.28} C_VEL
LIN {X 0,Y 379.886,Z 342.146,A -85,B 0,C 180,E1 -12259.198,E2 -12259.198} C_VEL
LIN {X 0,Y 376.215,Z 331.45,A -85,B 0,C 180,E1 -12260.004,E2 -12260.004} C_VEL
LIN {X 0,Y 376.392,Z 324.491,A -85,B 0,C 180,E1 -12264.254,E2 -12264.254} C_VEL
LIN {X 0,Y 376.575,Z 318.566,A -85,B 0,C 180,E1 -12267.812,E2 -12267.812} C_VEL
LIN {X 0,Y 376.935,Z 313.201,A -85,B 0,C 180,E1 -12270.943,E2 -12270.943} C_VEL
LIN {X 0,Y 377.104,Z 309.647,A -85,B 0,C 180,E1 -12273.001,E2 -12273.001} C_VEL
LIN {X 0,Y 376.626,Z 305.797,A -85,B 0,C 180,E1 -12275.343,E2 -12275.343} C_VEL
LIN {X 0,Y 375.949,Z 302.657,A -85,B 0,C 180,E1 -12277.413,E2 -12277.413} C_VEL
LIN {X 0,Y 375.94,Z 302.657,A -85,B 0,C 180,E1 -12280.867,E2 -12280.867} C_VEL
LIN {X 0,Y 375.99,Z 302.737,A -85,B 0,C 180,E1 -12283.757,E2 -12283.757} C_VEL
LIN {X 0,Y 377.356,Z 309.979,A -85,B 0,C 180,E1 -12287.278,E2 -12287.278} C_VEL
LIN {X 0,Y 379.028,Z 318.335,A -85,B 0,C 180,E1 -12291.148,E2 -12291.148} C_VEL
LIN {X 0,Y 379.584,Z 323.075,A -85,B 0,C 180,E1 -12293.225,E2 -12293.225} C_VEL
LIN {X 0,Y 379.033,Z 328.755,A -85,B 0,C 180,E1 -12295.561,E2 -12295.561} C_VEL
LIN {X 0,Y 378.12,Z 338.109,A -85,B 0,C 180,E1 -12299.301,E2 -12299.301} C_VEL
LIN {X 0,Y 377.125,Z 348.774,A -85,B 0,C 180,E1 -12303.447,E2 -12303.447} C_VEL
LIN {X 0,Y 376.433,Z 357.903,A -85,B 0,C 180,E1 -12306.917,E2 -12306.917} C_VEL
LIN {X 0,Y 375.779,Z 367.793,A -85,B 0,C 180,E1 -12310.612,E2 -12310.612} C_VEL
LIN {X 0,Y 375.759,Z 367.982,A -85,B 0,C 180,E1 -12310.682,E2 -12310.682} C_VEL
LIN {X 0,Y 378.496,Z 387.613,A -85,B 0,C 180,E1 -12311.676,E2 -12311.676} C_VEL
LIN {X 0,Y 379.861,Z 399.445,A -85,B 0,C 180,E1 -12312.45,E2 -12312.45} C_VEL
LIN {X 0,Y 380.109,Z 404.035,A -85,B 0,C 180,E1 -12312.793,E2 -12312.793} C_VEL
LIN {X 0,Y 379.016,Z 416.557,A -85,B 0,C 180,E1 -12313.851,E2 -12313.851} C_VEL
LIN {X 0,Y 378.072,Z 426.615,A -85,B 0,C 180,E1 -12314.915,E2 -12314.915} C_VEL
LIN {X 0,Y 377.245,Z 436.945,A -85,B 0,C 180,E1 -12316.259,E2 -12316.259} C_VEL
LIN {X 0,Y 376.444,Z 445.431,A -85,B 0,C 180,E1 -12317.602,E2 -12317.602} C_VEL
LIN {X 0,Y 375.669,Z 453.689,A -85,B 0,C 180,E1 -12319.218,E2 -12319.218} C_VEL
LIN {X 0,Y 375.233,Z 460.336,A -85,B 0,C 180,E1 -12320.839,E2 -12320.839} C_VEL
LIN {X 0,Y 374.889,Z 465.613,A -85,B 0,C 180,E1 -12322.459,E2 -12322.459} C_VEL
LIN {X 0,Y 374.733,Z 469.684,A -85,B 0,C 180,E1 -12324.054,E2 -12324.054} C_VEL
LIN {X 0,Y 374.627,Z 472.888,A -85,B 0,C 180,E1 -12325.696,E2 -12325.696} C_VEL
LIN {X 0,Y 374.658,Z 474.408,A -85,B 0,C 180,E1 -12326.774,E2 -12326.774} C_VEL
LIN {X 0,Y 374.692,Z 475.486,A -85,B 0,C 180,E1 -12327.85,E2 -12327.85} C_VEL
LIN {X 0,Y 374.754,Z 476.158,A -85,B 0,C 180,E1 -12328.925,E2 -12328.925} C_VEL
LIN {X 0,Y 374.748,Z 476.375,A -85,B 0,C 180,E1 -12330,E2 -12330} C_VEL
LIN {X 0,Y 374.746,Z 476.147,A -85,B 0,C 180,E1 -12331.075,E2 -12331.075} C_VEL
LIN {X 0,Y 374.705,Z 475.509,A -85,B 0,C 180,E1 -12332.15,E2 -12332.15} C_VEL
LIN {X 0,Y 374.642,Z 474.432,A -85,B 0,C 180,E1 -12333.226,E2 -12333.226} C_VEL
LIN {X 0,Y 374.639,Z 472.882,A -85,B 0,C 180,E1 -12334.303,E2 -12334.303} C_VEL
LIN {X 0,Y 374.731,Z 469.679,A -85,B 0,C 180,E1 -12335.945,E2 -12335.945} C_VEL
LIN {X 0,Y 374.887,Z 465.623,A -85,B 0,C 180,E1 -12337.541,E2 -12337.541} C_VEL
LIN {X 0,Y 375.276,Z 459.32,A -85,B 0,C 180,E1 -12339.431,E2 -12339.431} C_VEL
LIN {X 0,Y 375.79,Z 452.447,A -85,B 0,C 180,E1 -12341.052,E2 -12341.052} C_VEL
LIN {X 0,Y 376.444,Z 445.418,A -85,B 0,C 180,E1 -12342.398,E2 -12342.398} C_VEL
LIN {X 0,Y 377.252,Z 436.925,A -85,B 0,C 180,E1 -12343.741,E2 -12343.741} C_VEL
LIN {X 0,Y 378.182,Z 425.904,A -85,B 0,C 180,E1 -12345.218,E2 -12345.218} C_VEL
LIN {X 0,Y 379.297,Z 414.916,A -85,B 0,C 180,E1 -12346.414,E2 -12346.414} C_VEL
LIN {X 0,Y 380.362,Z 402.866,A -85,B 0,C 180,E1 -12347.473,E2 -12347.473} C_VEL
LIN {X 0,Y 379.358,Z 390.657,A -85,B 0,C 180,E1 -12348.436,E2 -12348.436} C_VEL
LIN {X 0,Y 378.234,Z 377.518,A -85,B 0,C 180,E1 -12349.261,E2 -12349.261} C_VEL
LIN {X 0,Y 376.003,Z 365.488,A -85,B 0,C 180,E1 -12349.931,E2 -12349.931} C_VEL
LIN {X 0,Y 375.738,Z 363.559,A -85,B 0,C 180,E1 -12350.031,E2 -12350.031} C_VEL
LIN {X 0,Y 376.36,Z 353.468,A -85,B 0,C 180,E1 -12353.793,E2 -12353.793} C_VEL
LIN {X 0,Y 376.975,Z 344.781,A -85,B 0,C 180,E1 -12357.178,E2 -12357.178} C_VEL
LIN {X 0,Y 377.795,Z 336.3,A -85,B 0,C 180,E1 -12360.683,E2 -12360.683} C_VEL
LIN {X 0,Y 378.699,Z 329.236,A -85,B 0,C 180,E1 -12363.831,E2 -12363.831} C_VEL
LIN {X 0,Y 379.534,Z 324.078,A -85,B 0,C 180,E1 -12366.339,E2 -12366.339} C_VEL
LIN {X 0,Y 379.381,Z 320.626,A -85,B 0,C 180,E1 -12368.275,E2 -12368.275} C_VEL
LIN {X 0,Y 378.8,Z 317.218,A -85,B 0,C 180,E1 -12370.494,E2 -12370.494} C_VEL
LIN {X 0,Y 378.061,Z 313.372,A -85,B 0,C 180,E1 -12373.532,E2 -12373.532} C_VEL
LIN {X 0,Y 377.508,Z 310.474,A -85,B 0,C 180,E1 -12376.557,E2 -12376.557} C_VEL
LIN {X 0,Y 377.096,Z 308.387,A -85,B 0,C 180,E1 -12379.829,E2 -12379.829} C_VEL
LIN {X 0,Y 376.942,Z 307.553,A -85,B 0,C 180,E1 -12382.028,E2 -12382.028} C_VEL
LIN {X 0,Y 376.799,Z 307.08,A -85,B 0,C 180,E1 -12385.153,E2 -12385.153} C_VEL
LIN {X 0,Y 376.784,Z 307.309,A -85,B 0,C 180,E1 -12388.515,E2 -12388.515} C_VEL
LIN {X 0,Y 376.932,Z 308.268,A -85,B 0,C 180,E1 -12392.216,E2 -12392.216} C_VEL
LIN {X 0,Y 377.003,Z 309.214,A -85,B 0,C 180,E1 -12394.611,E2 -12394.611} C_VEL
LIN {X 0,Y 376.927,Z 310.372,A -85,B 0,C 180,E1 -12396.949,E2 -12396.949} C_VEL
LIN {X 0,Y 376.768,Z 312.207,A -85,B 0,C 180,E1 -12400.124,E2 -12400.124} C_VEL
LIN {X 0,Y 381.853,Z 325.061,A -85,B 0,C 180,E1 -12401.225,E2 -12401.225} C_VEL
LIN {X 0,Y 383.612,Z 330.955,A -85,B 0,C 180,E1 -12401.751,E2 -12401.751} C_VEL
LIN {X 0,Y 382.763,Z 343.2,A -85,B 0,C 180,E1 -12402.641,E2 -12402.641} C_VEL
LIN {X 0,Y 381.65,Z 355.777,A -85,B 0,C 180,E1 -12403.813,E2 -12403.813} C_VEL
LIN {X 0,Y 380.642,Z 365.983,A -85,B 0,C 180,E1 -12405.02,E2 -12405.02} C_VEL
LIN {X 0,Y 379.598,Z 375.203,A -85,B 0,C 180,E1 -12406.346,E2 -12406.346} C_VEL
LIN {X 0,Y 378.785,Z 382.816,A -85,B 0,C 180,E1 -12407.68,E2 -12407.68} C_VEL
LIN {X 0,Y 377.791,Z 390.28,A -85,B 0,C 180,E1 -12409.279,E2 -12409.279} C_VEL
LIN {X 0,Y 377.053,Z 396.77,A -85,B 0,C 180,E1 -12411.073,E2 -12411.073} C_VEL
LIN {X 0,Y 376.397,Z 400.836,A -85,B 0,C 180,E1 -12412.49,E2 -12412.49} C_VEL
LIN {X 0,Y 376.104,Z 403.309,A -85,B 0,C 180,E1 -12413.563,E2 -12413.563} C_VEL
LIN {X 0,Y 375.951,Z 405.273,A -85,B 0,C 180,E1 -12414.637,E2 -12414.637} C_VEL
LIN {X 0,Y 375.655,Z 406.79,A -85,B 0,C 180,E1 -12415.708,E2 -12415.708} C_VEL
LIN {X 0,Y 375.335,Z 407.899,A -85,B 0,C 180,E1 -12416.78,E2 -12416.78} C_VEL
LIN {X 0,Y 375.111,Z 408.574,A -85,B 0,C 180,E1 -12417.853,E2 -12417.853} C_VEL
LIN {X 0,Y 374.998,Z 408.786,A -85,B 0,C 180,E1 -12418.926,E2 -12418.926} C_VEL
LIN {X 0,Y 374.953,Z 408.592,A -85,B 0,C 180,E1 -12420,E2 -12420} C_VEL
LIN {X 0,Y 374.974,Z 407.992,A -85,B 0,C 180,E1 -12421.074,E2 -12421.074} C_VEL
LIN {X 0,Y 375.089,Z 406.929,A -85,B 0,C 180,E1 -12422.148,E2 -12422.148} C_VEL
LIN {X 0,Y 375.228,Z 405.438,A -85,B 0,C 180,E1 -12423.221,E2 -12423.221} C_VEL
LIN {X 0,Y 375.477,Z 402.378,A -85,B 0,C 180,E1 -12424.832,E2 -12424.832} C_VEL
LIN {X 0,Y 375.536,Z 398.258,A -85,B 0,C 180,E1 -12426.447,E2 -12426.447} C_VEL
LIN {X 0,Y 375.965,Z 392.042,A -85,B 0,C 180,E1 -12428.303,E2 -12428.303} C_VEL
LIN {X 0,Y 376.424,Z 384.995,A -85,B 0,C 180,E1 -12429.945,E2 -12429.945} C_VEL
LIN {X 0,Y 377.035,Z 376.413,A -85,B 0,C 180,E1 -12431.559,E2 -12431.559} C_VEL
LIN {X 0,Y 377.639,Z 367.664,A -85,B 0,C 180,E1 -12432.904,E2 -12432.904} C_VEL
LIN {X 0,Y 378.395,Z 356.931,A -85,B 0,C 180,E1 -12434.247,E2 -12434.247} C_VEL
LIN {X 0,Y 379.052,Z 344.94,A -85,B 0,C 180,E1 -12435.46,E2 -12435.46} C_VEL
LIN {X 0,Y 379.657,Z 333.165,A -85,B 0,C 180,E1 -12436.398,E2 -12436.398} C_VEL
LIN {X 0,Y 380.061,Z 323.748,A -85,B 0,C 180,E1 -12437.002,E2 -12437.002} C_VEL
LIN {X 0,Y 376.889,Z 310.099,A -85,B 0,C 180,E1 -12437.802,E2 -12437.802} C_VEL
LIN {X 0,Y 375.246,Z 303.007,A -85,B 0,C 180,E1 -12438.145,E2 -12438.145} C_VEL
LIN {X 0,Y 375.268,Z 302.744,A -85,B 0,C 180,E1 -12438.565,E2 -12438.565} C_VEL
LIN {X 0,Y 375.64,Z 302.69,A -85,B 0,C 180,E1 -12441.974,E2 -12441.974} C_VEL
LIN {X 0,Y 375.842,Z 302.67,A -85,B 0,C 180,E1 -12444.292,E2 -12444.292} C_VEL
LIN {X 0,Y 375.96,Z 302.648,A -85,B 0,C 180,E1 -12446.657,E2 -12446.657} C_VEL
LIN {X 0,Y 375.961,Z 302.653,A -85,B 0,C 180,E1 -12449.08,E2 -12449.08} C_VEL
LIN {X 0,Y 375.953,Z 302.656,A -85,B 0,C 180,E1 -12452.828,E2 -12452.828} C_VEL
LIN {X 0,Y 375.96,Z 302.647,A -85,B 0,C 180,E1 -12455.415,E2 -12455.415} C_VEL
LIN {X 0,Y 375.976,Z 302.653,A -85,B 0,C 180,E1 -12458.27,E2 -12458.27} C_VEL
LIN {X 0,Y 375.937,Z 302.66,A -85,B 0,C 180,E1 -12461.601,E2 -12461.601} C_VEL
LIN {X 0,Y 375.93,Z 302.656,A -85,B 0,C 180,E1 -12465.268,E2 -12465.268} C_VEL
LIN {X 0,Y 375.937,Z 302.656,A -85,B 0,C 180,E1 -12468.399,E2 -12468.399} C_VEL
LIN {X 0,Y 375.975,Z 302.654,A -85,B 0,C 180,E1 -12471.73,E2 -12471.73} C_VEL
LIN {X 0,Y 375.878,Z 302.668,A -85,B 0,C 180,E1 -12474.576,E2 -12474.576} C_VEL
LIN {X 0,Y 375.881,Z 302.868,A -85,B 0,C 180,E1 -12476.203,E2 -12476.203} C_VEL
LIN {X 0,Y 375.585,Z 308.293,A -85,B 0,C 180,E1 -12479.653,E2 -12479.653} C_VEL
LIN {X 0,Y 375.514,Z 312.122,A -85,B 0,C 180,E1 -12482.102,E2 -12482.102} C_VEL
LIN {X 0,Y 375.401,Z 317.874,A -85,B 0,C 180,E1 -12485.678,E2 -12485.678} C_VEL
LIN {X 0,Y 375.411,Z 324.181,A -85,B 0,C 180,E1 -12489.398,E2 -12489.398} C_VEL
LIN {X 0,Y 375.385,Z 326.751,A -85,B 0,C 180,E1 -12490.816,E2 -12490.816} C_VEL
LIN {X 0,Y 379.003,Z 340.31,A -85,B 0,C 180,E1 -12491.468,E2 -12491.468} C_VEL
LIN {X 0,Y 381.575,Z 352.224,A -85,B 0,C 180,E1 -12492.213,E2 -12492.213} C_VEL
LIN {X 0,Y 380.997,Z 363.532,A -85,B 0,C 180,E1 -12492.972,E2 -12492.972} C_VEL
LIN {X 0,Y 380.213,Z 374.372,A -85,B 0,C 180,E1 -12493.903,E2 -12493.903} C_VEL
LIN {X 0,Y 379.346,Z 385.45,A -85,B 0,C 180,E1 -12495.104,E2 -12495.104} C_VEL
LIN {X 0,Y 378.486,Z 394.401,A -85,B 0,C 180,E1 -12496.305,E2 -12496.305} C_VEL
LIN {X 0,Y 377.472,Z 404.025,A -85,B 0,C 180,E1 -12497.909,E2 -12497.909} C_VEL
LIN {X 0,Y 376.675,Z 411.755,A -85,B 0,C 180,E1 -12499.519,E2 -12499.519} C_VEL
LIN {X 0,Y 376.076,Z 416.978,A -85,B 0,C 180,E1 -12500.86,E2 -12500.86} C_VEL
LIN {X 0,Y 375.528,Z 422.694,A -85,B 0,C 180,E1 -12502.701,E2 -12502.701} C_VEL
LIN {X 0,Y 375.051,Z 427.086,A -85,B 0,C 180,E1 -12504.624,E2 -12504.624} C_VEL
LIN {X 0,Y 375.006,Z 428.928,A -85,B 0,C 180,E1 -12505.701,E2 -12505.701} C_VEL
LIN {X 0,Y 374.962,Z 430.334,A -85,B 0,C 180,E1 -12506.777,E2 -12506.777} C_VEL
LIN {X 0,Y 374.694,Z 431.942,A -85,B 0,C 180,E1 -12508.925,E2 -12508.925} C_VEL
LIN {X 0,Y 374.674,Z 432.176,A -85,B 0,C 180,E1 -12510,E2 -12510} C_VEL
LIN {X 0,Y 374.802,Z 431.399,A -85,B 0,C 180,E1 -12512.149,E2 -12512.149} C_VEL
LIN {X 0,Y 374.958,Z 430.433,A -85,B 0,C 180,E1 -12513.223,E2 -12513.223} C_VEL
LIN {X 0,Y 374.979,Z 429.084,A -85,B 0,C 180,E1 -12514.299,E2 -12514.299} C_VEL
LIN {X 0,Y 375.169,Z 426.234,A -85,B 0,C 180,E1 -12515.914,E2 -12515.914} C_VEL
LIN {X 0,Y 375.561,Z 422.356,A -85,B 0,C 180,E1 -12517.527,E2 -12517.527} C_VEL
LIN {X 0,Y 376.032,Z 417.335,A -85,B 0,C 180,E1 -12519.141,E2 -12519.141} C_VEL
LIN {X 0,Y 376.761,Z 410.99,A -85,B 0,C 180,E1 -12520.751,E2 -12520.751} C_VEL
LIN {X 0,Y 377.576,Z 403.106,A -85,B 0,C 180,E1 -12522.36,E2 -12522.36} C_VEL
LIN {X 0,Y 378.435,Z 395.044,A -85,B 0,C 180,E1 -12523.697,E2 -12523.697} C_VEL
LIN {X 0,Y 379.417,Z 385.144,A -85,B 0,C 180,E1 -12525.03,E2 -12525.03} C_VEL
LIN {X 0,Y 380.115,Z 375.371,A -85,B 0,C 180,E1 -12526.101,E2 -12526.101} C_VEL
LIN {X 0,Y 380.958,Z 364.76,A -85,B 0,C 180,E1 -12527.03,E2 -12527.03} C_VEL
LIN {X 0,Y 381.645,Z 352.721,A -85,B 0,C 180,E1 -12527.853,E2 -12527.853} C_VEL
LIN {X 0,Y 379.21,Z 341.013,A -85,B 0,C 180,E1 -12528.593,E2 -12528.593} C_VEL
LIN {X 0,Y 376.097,Z 329.422,A -85,B 0,C 180,E1 -12529.174,E2 -12529.174} C_VEL
LIN {X 0,Y 375.403,Z 327.575,A -85,B 0,C 180,E1 -12529.357,E2 -12529.357} C_VEL
LIN {X 0,Y 373.876,Z 325.898,A -85,B 0,C 180,E1 -12529.874,E2 -12529.874} C_VEL
LIN {X 0,Y 370.209,Z 323.595,A -85,B 0,C 180,E1 -12531.623,E2 -12531.623} C_VEL
LIN {X 0,Y 368.624,Z 321.355,A -85,B 0,C 180,E1 -12532.975,E2 -12532.975} C_VEL
LIN {X 0,Y 368.379,Z 320.193,A -85,B 0,C 180,E1 -12533.66,E2 -12533.66} C_VEL
LIN {X 0,Y 368.429,Z 314.411,A -85,B 0,C 180,E1 -12537.246,E2 -12537.246} C_VEL
LIN {X 0,Y 368.578,Z 308.689,A -85,B 0,C 180,E1 -12540.901,E2 -12540.901} C_VEL
LIN {X 0,Y 368.822,Z 303.546,A -85,B 0,C 180,E1 -12544.203,E2 -12544.203} C_VEL
LIN {X 0,Y 368.899,Z 303.535,A -85,B 0,C 180,E1 -12547.564,E2 -12547.564} C_VEL
LIN {X 0,Y 368.913,Z 303.534,A -85,B 0,C 180,E1 -12550.37,E2 -12550.37} C_VEL
LIN {X 0,Y 368.885,Z 303.538,A -85,B 0,C 180,E1 -12553.616,E2 -12553.616} C_VEL
LIN {X 0,Y 368.888,Z 303.537,A -85,B 0,C 180,E1 -12556.696,E2 -12556.696} C_VEL
LIN {X 0,Y 368.914,Z 303.532,A -85,B 0,C 180,E1 -12559.643,E2 -12559.643} C_VEL
LIN {X 0,Y 368.873,Z 303.538,A -85,B 0,C 180,E1 -12563.151,E2 -12563.151} C_VEL
LIN {X 0,Y 368.723,Z 303.557,A -85,B 0,C 180,E1 -12566.444,E2 -12566.444} C_VEL
LIN {X 0,Y 368.618,Z 303.582,A -85,B 0,C 180,E1 -12567.024,E2 -12567.024} C_VEL
LIN {X 0,Y 368.325,Z 310.76,A -85,B 0,C 180,E1 -12571.509,E2 -12571.509} C_VEL
